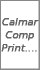
VISUALIZATION _VISU_CTsFlow  // 40x70
VAR_IN_OUT
	m_Inst  : FB_PrintOverview;
END_VAR
    Frame (0,0 40x70), invisible if: m_Inst.aCTV[30]._hidden
        shows CalmarCompPrint._VISU_ContainerView(m_Inst := m_Inst.aCTV[30])
        p3560616238: m_Inst.aCTV[30]._posX
        p2738717112: m_Inst.aCTV[30]._posY
    Frame (0,0 40x70), invisible if: m_Inst.aCTV[31]._hidden
        shows CalmarCompPrint._VISU_ContainerView(m_Inst := m_Inst.aCTV[31])
        p3560616238: m_Inst.aCTV[31]._posX
        p2738717112: m_Inst.aCTV[31]._posY
    Frame (0,0 40x70), invisible if: m_Inst.aCTV[32]._hidden
        shows CalmarCompPrint._VISU_ContainerView(m_Inst := m_Inst.aCTV[32])
        p3560616238: m_Inst.aCTV[32]._posX
        p2738717112: m_Inst.aCTV[32]._posY
    Frame (0,0 40x70), invisible if: m_Inst.aCTV[33]._hidden
        shows CalmarCompPrint._VISU_ContainerView(m_Inst := m_Inst.aCTV[33])
        p3560616238: m_Inst.aCTV[33]._posX
        p2738717112: m_Inst.aCTV[33]._posY
    Frame (0,0 40x70), invisible if: m_Inst.aCTV[34]._hidden
        shows CalmarCompPrint._VISU_ContainerView(m_Inst := m_Inst.aCTV[34])
        p3560616238: m_Inst.aCTV[34]._posX
        p2738717112: m_Inst.aCTV[34]._posY
    Frame (0,0 40x70), invisible if: m_Inst.aCTV[35]._hidden
        shows CalmarCompPrint._VISU_ContainerView(m_Inst := m_Inst.aCTV[35])
        p3560616238: m_Inst.aCTV[35]._posX
        p2738717112: m_Inst.aCTV[35]._posY
    Frame (0,0 40x70), invisible if: m_Inst.aCTV[36]._hidden
        shows CalmarCompPrint._VISU_ContainerView(m_Inst := m_Inst.aCTV[36])
        p3560616238: m_Inst.aCTV[36]._posX
        p2738717112: m_Inst.aCTV[36]._posY
    Frame (0,0 40x70), invisible if: m_Inst.aCTV[37]._hidden
        shows CalmarCompPrint._VISU_ContainerView(m_Inst := m_Inst.aCTV[37])
        p3560616238: m_Inst.aCTV[37]._posX
        p2738717112: m_Inst.aCTV[37]._posY
    Frame (0,0 40x70), invisible if: m_Inst.aCTV[38]._hidden
        shows CalmarCompPrint._VISU_ContainerView(m_Inst := m_Inst.aCTV[38])
        p3560616238: m_Inst.aCTV[38]._posX
        p2738717112: m_Inst.aCTV[38]._posY
    Frame (0,0 40x70), invisible if: m_Inst.aCTV[39]._hidden
        shows CalmarCompPrint._VISU_ContainerView(m_Inst := m_Inst.aCTV[39])
        p3560616238: m_Inst.aCTV[39]._posX
        p2738717112: m_Inst.aCTV[39]._posY
    Frame (0,0 40x70), invisible if: m_Inst.aCTV[10]._hidden
        shows CalmarCompPrint._VISU_ContainerView(m_Inst := m_Inst.aCTV[10])
        p3560616238: m_Inst.aCTV[10]._posX
        p2738717112: m_Inst.aCTV[10]._posY
    Frame (0,0 40x70), invisible if: m_Inst.aCTV[11]._hidden
        shows CalmarCompPrint._VISU_ContainerView(m_Inst := m_Inst.aCTV[11])
        p3560616238: m_Inst.aCTV[11]._posX
        p2738717112: m_Inst.aCTV[11]._posY
    Frame (0,0 40x70), invisible if: m_Inst.aCTV[12]._hidden
        shows CalmarCompPrint._VISU_ContainerView(m_Inst := m_Inst.aCTV[12])
        p3560616238: m_Inst.aCTV[12]._posX
        p2738717112: m_Inst.aCTV[12]._posY
    Frame (0,0 40x70), invisible if: m_Inst.aCTV[13]._hidden
        shows CalmarCompPrint._VISU_ContainerView(m_Inst := m_Inst.aCTV[13])
        p3560616238: m_Inst.aCTV[13]._posX
        p2738717112: m_Inst.aCTV[13]._posY
    Frame (0,0 40x70), invisible if: m_Inst.aCTV[14]._hidden
        shows CalmarCompPrint._VISU_ContainerView(m_Inst := m_Inst.aCTV[14])
        p3560616238: m_Inst.aCTV[14]._posX
        p2738717112: m_Inst.aCTV[14]._posY
    Frame (0,0 40x70), invisible if: m_Inst.aCTV[15]._hidden
        shows CalmarCompPrint._VISU_ContainerView(m_Inst := m_Inst.aCTV[15])
        p3560616238: m_Inst.aCTV[15]._posX
        p2738717112: m_Inst.aCTV[15]._posY
    Frame (0,0 40x70), invisible if: m_Inst.aCTV[16]._hidden
        shows CalmarCompPrint._VISU_ContainerView(m_Inst := m_Inst.aCTV[16])
        p3560616238: m_Inst.aCTV[16]._posX
        p2738717112: m_Inst.aCTV[16]._posY
    Frame (0,0 40x70), invisible if: m_Inst.aCTV[17]._hidden
        shows CalmarCompPrint._VISU_ContainerView(m_Inst := m_Inst.aCTV[17])
        p3560616238: m_Inst.aCTV[17]._posX
        p2738717112: m_Inst.aCTV[17]._posY
    Frame (0,0 40x70), invisible if: m_Inst.aCTV[18]._hidden
        shows CalmarCompPrint._VISU_ContainerView(m_Inst := m_Inst.aCTV[18])
        p3560616238: m_Inst.aCTV[18]._posX
        p2738717112: m_Inst.aCTV[18]._posY
    Frame (0,0 40x70), invisible if: m_Inst.aCTV[19]._hidden
        shows CalmarCompPrint._VISU_ContainerView(m_Inst := m_Inst.aCTV[19])
        p3560616238: m_Inst.aCTV[19]._posX
        p2738717112: m_Inst.aCTV[19]._posY
    Frame (0,0 40x70), invisible if: m_Inst.aCTV[20]._hidden
        shows CalmarCompPrint._VISU_ContainerView(m_Inst := m_Inst.aCTV[20])
        p3560616238: m_Inst.aCTV[20]._posX
        p2738717112: m_Inst.aCTV[20]._posY
    Frame (0,0 40x70), invisible if: m_Inst.aCTV[21]._hidden
        shows CalmarCompPrint._VISU_ContainerView(m_Inst := m_Inst.aCTV[21])
        p3560616238: m_Inst.aCTV[21]._posX
        p2738717112: m_Inst.aCTV[21]._posY
    Frame (0,0 40x70), invisible if: m_Inst.aCTV[22]._hidden
        shows CalmarCompPrint._VISU_ContainerView(m_Inst := m_Inst.aCTV[22])
        p3560616238: m_Inst.aCTV[22]._posX
        p2738717112: m_Inst.aCTV[22]._posY
    Frame (0,0 40x70), invisible if: m_Inst.aCTV[23]._hidden
        shows CalmarCompPrint._VISU_ContainerView(m_Inst := m_Inst.aCTV[23])
        p3560616238: m_Inst.aCTV[23]._posX
        p2738717112: m_Inst.aCTV[23]._posY
    Frame (0,0 40x70), invisible if: m_Inst.aCTV[24]._hidden
        shows CalmarCompPrint._VISU_ContainerView(m_Inst := m_Inst.aCTV[24])
        p3560616238: m_Inst.aCTV[24]._posX
        p2738717112: m_Inst.aCTV[24]._posY
    Frame (0,0 40x70), invisible if: m_Inst.aCTV[25]._hidden
        shows CalmarCompPrint._VISU_ContainerView(m_Inst := m_Inst.aCTV[25])
        p3560616238: m_Inst.aCTV[25]._posX
        p2738717112: m_Inst.aCTV[25]._posY
    Frame (0,0 40x70), invisible if: m_Inst.aCTV[26]._hidden
        shows CalmarCompPrint._VISU_ContainerView(m_Inst := m_Inst.aCTV[26])
        p3560616238: m_Inst.aCTV[26]._posX
        p2738717112: m_Inst.aCTV[26]._posY
    Frame (0,0 40x70), invisible if: m_Inst.aCTV[27]._hidden
        shows CalmarCompPrint._VISU_ContainerView(m_Inst := m_Inst.aCTV[27])
        p3560616238: m_Inst.aCTV[27]._posX
        p2738717112: m_Inst.aCTV[27]._posY
    Frame (0,0 40x70), invisible if: m_Inst.aCTV[28]._hidden
        shows CalmarCompPrint._VISU_ContainerView(m_Inst := m_Inst.aCTV[28])
        p3560616238: m_Inst.aCTV[28]._posX
        p2738717112: m_Inst.aCTV[28]._posY
    Frame (0,0 40x70), invisible if: m_Inst.aCTV[29]._hidden
        shows CalmarCompPrint._VISU_ContainerView(m_Inst := m_Inst.aCTV[29])
        p3560616238: m_Inst.aCTV[29]._posX
        p2738717112: m_Inst.aCTV[29]._posY
    Frame (0,0 40x70), invisible if: m_Inst.aCTV[40]._hidden
        shows CalmarCompPrint._VISU_ContainerView(m_Inst := m_Inst.aCTV[40])
        p3560616238: m_Inst.aCTV[40]._posX
        p2738717112: m_Inst.aCTV[40]._posY
    Frame (0,0 40x70), invisible if: m_Inst.aCTV[41]._hidden
        shows CalmarCompPrint._VISU_ContainerView(m_Inst := m_Inst.aCTV[41])
        p3560616238: m_Inst.aCTV[41]._posX
        p2738717112: m_Inst.aCTV[41]._posY
    Frame (0,0 40x70), invisible if: m_Inst.aCTV[42]._hidden
        shows CalmarCompPrint._VISU_ContainerView(m_Inst := m_Inst.aCTV[42])
        p3560616238: m_Inst.aCTV[42]._posX
        p2738717112: m_Inst.aCTV[42]._posY
    Frame (0,0 40x70), invisible if: m_Inst.aCTV[43]._hidden
        shows CalmarCompPrint._VISU_ContainerView(m_Inst := m_Inst.aCTV[43])
        p3560616238: m_Inst.aCTV[43]._posX
        p2738717112: m_Inst.aCTV[43]._posY
    Frame (0,0 40x70), invisible if: m_Inst.aCTV[44]._hidden
        shows CalmarCompPrint._VISU_ContainerView(m_Inst := m_Inst.aCTV[44])
        p3560616238: m_Inst.aCTV[44]._posX
        p2738717112: m_Inst.aCTV[44]._posY
    Frame (0,0 40x70), invisible if: m_Inst.aCTV[45]._hidden
        shows CalmarCompPrint._VISU_ContainerView(m_Inst := m_Inst.aCTV[45])
        p3560616238: m_Inst.aCTV[45]._posX
        p2738717112: m_Inst.aCTV[45]._posY
    Frame (0,0 40x70), invisible if: m_Inst.aCTV[46]._hidden
        shows CalmarCompPrint._VISU_ContainerView(m_Inst := m_Inst.aCTV[46])
        p3560616238: m_Inst.aCTV[46]._posX
        p2738717112: m_Inst.aCTV[46]._posY
    Frame (0,0 40x70), invisible if: m_Inst.aCTV[47]._hidden
        shows CalmarCompPrint._VISU_ContainerView(m_Inst := m_Inst.aCTV[47])
        p3560616238: m_Inst.aCTV[47]._posX
        p2738717112: m_Inst.aCTV[47]._posY
    Frame (0,0 40x70), invisible if: m_Inst.aCTV[48]._hidden
        shows CalmarCompPrint._VISU_ContainerView(m_Inst := m_Inst.aCTV[48])
        p3560616238: m_Inst.aCTV[48]._posX
        p2738717112: m_Inst.aCTV[48]._posY
    Frame (0,0 40x70), invisible if: m_Inst.aCTV[49]._hidden
        shows CalmarCompPrint._VISU_ContainerView(m_Inst := m_Inst.aCTV[49])
        p3560616238: m_Inst.aCTV[49]._posX
        p2738717112: m_Inst.aCTV[49]._posY
    Frame (0,0 40x70), invisible if: m_Inst.aCTV[49]._hidden
        shows CalmarCompPrint._VISU_ContainerView(m_Inst := m_Inst.aCTV[49])
        p3560616238: m_Inst.aCTV[49]._posX
        p2738717112: m_Inst.aCTV[49]._posY
    Frame (0,0 40x70), invisible if: m_Inst.aCTV[1]._hidden
        shows CalmarCompPrint._VISU_ContainerView(m_Inst := m_Inst.aCTV[1])
        p3560616238: m_Inst.aCTV[1]._posX
        p2738717112: m_Inst.aCTV[1]._posY
    Frame (0,0 40x70), invisible if: m_Inst.aCTV[2]._hidden
        shows CalmarCompPrint._VISU_ContainerView(m_Inst := m_Inst.aCTV[2])
        p3560616238: m_Inst.aCTV[2]._posX
        p2738717112: m_Inst.aCTV[2]._posY
    Frame (0,0 40x70), invisible if: m_Inst.aCTV[3]._hidden
        shows CalmarCompPrint._VISU_ContainerView(m_Inst := m_Inst.aCTV[3])
        p3560616238: m_Inst.aCTV[3]._posX
        p2738717112: m_Inst.aCTV[3]._posY
    Frame (0,0 40x70), invisible if: m_Inst.aCTV[4]._hidden
        shows CalmarCompPrint._VISU_ContainerView(m_Inst := m_Inst.aCTV[4])
        p3560616238: m_Inst.aCTV[4]._posX
        p2738717112: m_Inst.aCTV[4]._posY
    Frame (0,0 40x70), invisible if: m_Inst.aCTV[5]._hidden
        shows CalmarCompPrint._VISU_ContainerView(m_Inst := m_Inst.aCTV[5])
        p3560616238: m_Inst.aCTV[5]._posX
        p2738717112: m_Inst.aCTV[5]._posY
    Frame (0,0 40x70), invisible if: m_Inst.aCTV[6]._hidden
        shows CalmarCompPrint._VISU_ContainerView(m_Inst := m_Inst.aCTV[6])
        p3560616238: m_Inst.aCTV[6]._posX
        p2738717112: m_Inst.aCTV[6]._posY
    Frame (0,0 40x70), invisible if: m_Inst.aCTV[7]._hidden
        shows CalmarCompPrint._VISU_ContainerView(m_Inst := m_Inst.aCTV[7])
        p3560616238: m_Inst.aCTV[7]._posX
        p2738717112: m_Inst.aCTV[7]._posY
    Frame (0,0 40x70), invisible if: m_Inst.aCTV[8]._hidden
        shows CalmarCompPrint._VISU_ContainerView(m_Inst := m_Inst.aCTV[8])
        p3560616238: m_Inst.aCTV[8]._posX
        p2738717112: m_Inst.aCTV[8]._posY
    Frame (0,0 40x70), invisible if: m_Inst.aCTV[9]._hidden
        shows CalmarCompPrint._VISU_ContainerView(m_Inst := m_Inst.aCTV[9])
        p3560616238: m_Inst.aCTV[9]._posX
        p2738717112: m_Inst.aCTV[9]._posY
END_VISUALIZATION

// ---- POUs/Print/DefGrid/_VISU_Templates/_VISU_CTTrackerFlow.TcVIS
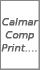
VISUALIZATION _VISU_CTTrackerFlow  // 40x70
VAR_IN_OUT
	m_Inst  : FB_CTTrackerView;
END_VAR
    Frame (0,0 40x70), invisible if: m_Inst.aCTV[30]._hidden
        shows CalmarCompPrint._VISU_ContainerView(m_Inst := m_Inst.aCTV[30])
        p3560616238: m_Inst.aCTV[30]._posX
        p2738717112: m_Inst.aCTV[30]._posY
    Frame (0,0 40x70), invisible if: m_Inst.aCTV[31]._hidden
        shows CalmarCompPrint._VISU_ContainerView(m_Inst := m_Inst.aCTV[31])
        p3560616238: m_Inst.aCTV[31]._posX
        p2738717112: m_Inst.aCTV[31]._posY
    Frame (0,0 40x70), invisible if: m_Inst.aCTV[32]._hidden
        shows CalmarCompPrint._VISU_ContainerView(m_Inst := m_Inst.aCTV[32])
        p3560616238: m_Inst.aCTV[32]._posX
        p2738717112: m_Inst.aCTV[32]._posY
    Frame (0,0 40x70), invisible if: m_Inst.aCTV[33]._hidden
        shows CalmarCompPrint._VISU_ContainerView(m_Inst := m_Inst.aCTV[33])
        p3560616238: m_Inst.aCTV[33]._posX
        p2738717112: m_Inst.aCTV[33]._posY
    Frame (0,0 40x70), invisible if: m_Inst.aCTV[34]._hidden
        shows CalmarCompPrint._VISU_ContainerView(m_Inst := m_Inst.aCTV[34])
        p3560616238: m_Inst.aCTV[34]._posX
        p2738717112: m_Inst.aCTV[34]._posY
    Frame (0,0 40x70), invisible if: m_Inst.aCTV[35]._hidden
        shows CalmarCompPrint._VISU_ContainerView(m_Inst := m_Inst.aCTV[35])
        p3560616238: m_Inst.aCTV[35]._posX
        p2738717112: m_Inst.aCTV[35]._posY
    Frame (0,0 40x70), invisible if: m_Inst.aCTV[36]._hidden
        shows CalmarCompPrint._VISU_ContainerView(m_Inst := m_Inst.aCTV[36])
        p3560616238: m_Inst.aCTV[36]._posX
        p2738717112: m_Inst.aCTV[36]._posY
    Frame (0,0 40x70), invisible if: m_Inst.aCTV[37]._hidden
        shows CalmarCompPrint._VISU_ContainerView(m_Inst := m_Inst.aCTV[37])
        p3560616238: m_Inst.aCTV[37]._posX
        p2738717112: m_Inst.aCTV[37]._posY
    Frame (0,0 40x70), invisible if: m_Inst.aCTV[38]._hidden
        shows CalmarCompPrint._VISU_ContainerView(m_Inst := m_Inst.aCTV[38])
        p3560616238: m_Inst.aCTV[38]._posX
        p2738717112: m_Inst.aCTV[38]._posY
    Frame (0,0 40x70), invisible if: m_Inst.aCTV[39]._hidden
        shows CalmarCompPrint._VISU_ContainerView(m_Inst := m_Inst.aCTV[39])
        p3560616238: m_Inst.aCTV[39]._posX
        p2738717112: m_Inst.aCTV[39]._posY
    Frame (0,0 40x70), invisible if: m_Inst.aCTV[10]._hidden
        shows CalmarCompPrint._VISU_ContainerView(m_Inst := m_Inst.aCTV[10])
        p3560616238: m_Inst.aCTV[10]._posX
        p2738717112: m_Inst.aCTV[10]._posY
    Frame (0,0 40x70), invisible if: m_Inst.aCTV[11]._hidden
        shows CalmarCompPrint._VISU_ContainerView(m_Inst := m_Inst.aCTV[11])
        p3560616238: m_Inst.aCTV[11]._posX
        p2738717112: m_Inst.aCTV[11]._posY
    Frame (0,0 40x70), invisible if: m_Inst.aCTV[12]._hidden
        shows CalmarCompPrint._VISU_ContainerView(m_Inst := m_Inst.aCTV[12])
        p3560616238: m_Inst.aCTV[12]._posX
        p2738717112: m_Inst.aCTV[12]._posY
    Frame (0,0 40x70), invisible if: m_Inst.aCTV[13]._hidden
        shows CalmarCompPrint._VISU_ContainerView(m_Inst := m_Inst.aCTV[13])
        p3560616238: m_Inst.aCTV[13]._posX
        p2738717112: m_Inst.aCTV[13]._posY
    Frame (0,0 40x70), invisible if: m_Inst.aCTV[14]._hidden
        shows CalmarCompPrint._VISU_ContainerView(m_Inst := m_Inst.aCTV[14])
        p3560616238: m_Inst.aCTV[14]._posX
        p2738717112: m_Inst.aCTV[14]._posY
    Frame (0,0 40x70), invisible if: m_Inst.aCTV[15]._hidden
        shows CalmarCompPrint._VISU_ContainerView(m_Inst := m_Inst.aCTV[15])
        p3560616238: m_Inst.aCTV[15]._posX
        p2738717112: m_Inst.aCTV[15]._posY
    Frame (0,0 40x70), invisible if: m_Inst.aCTV[16]._hidden
        shows CalmarCompPrint._VISU_ContainerView(m_Inst := m_Inst.aCTV[16])
        p3560616238: m_Inst.aCTV[16]._posX
        p2738717112: m_Inst.aCTV[16]._posY
    Frame (0,0 40x70), invisible if: m_Inst.aCTV[17]._hidden
        shows CalmarCompPrint._VISU_ContainerView(m_Inst := m_Inst.aCTV[17])
        p3560616238: m_Inst.aCTV[17]._posX
        p2738717112: m_Inst.aCTV[17]._posY
    Frame (0,0 40x70), invisible if: m_Inst.aCTV[18]._hidden
        shows CalmarCompPrint._VISU_ContainerView(m_Inst := m_Inst.aCTV[18])
        p3560616238: m_Inst.aCTV[18]._posX
        p2738717112: m_Inst.aCTV[18]._posY
    Frame (0,0 40x70), invisible if: m_Inst.aCTV[19]._hidden
        shows CalmarCompPrint._VISU_ContainerView(m_Inst := m_Inst.aCTV[19])
        p3560616238: m_Inst.aCTV[19]._posX
        p2738717112: m_Inst.aCTV[19]._posY
    Frame (0,0 40x70), invisible if: m_Inst.aCTV[20]._hidden
        shows CalmarCompPrint._VISU_ContainerView(m_Inst := m_Inst.aCTV[20])
        p3560616238: m_Inst.aCTV[20]._posX
        p2738717112: m_Inst.aCTV[20]._posY
    Frame (0,0 40x70), invisible if: m_Inst.aCTV[21]._hidden
        shows CalmarCompPrint._VISU_ContainerView(m_Inst := m_Inst.aCTV[21])
        p3560616238: m_Inst.aCTV[21]._posX
        p2738717112: m_Inst.aCTV[21]._posY
    Frame (0,0 40x70), invisible if: m_Inst.aCTV[22]._hidden
        shows CalmarCompPrint._VISU_ContainerView(m_Inst := m_Inst.aCTV[22])
        p3560616238: m_Inst.aCTV[22]._posX
        p2738717112: m_Inst.aCTV[22]._posY
    Frame (0,0 40x70), invisible if: m_Inst.aCTV[23]._hidden
        shows CalmarCompPrint._VISU_ContainerView(m_Inst := m_Inst.aCTV[23])
        p3560616238: m_Inst.aCTV[23]._posX
        p2738717112: m_Inst.aCTV[23]._posY
    Frame (0,0 40x70), invisible if: m_Inst.aCTV[24]._hidden
        shows CalmarCompPrint._VISU_ContainerView(m_Inst := m_Inst.aCTV[24])
        p3560616238: m_Inst.aCTV[24]._posX
        p2738717112: m_Inst.aCTV[24]._posY
    Frame (0,0 40x70), invisible if: m_Inst.aCTV[25]._hidden
        shows CalmarCompPrint._VISU_ContainerView(m_Inst := m_Inst.aCTV[25])
        p3560616238: m_Inst.aCTV[25]._posX
        p2738717112: m_Inst.aCTV[25]._posY
    Frame (0,0 40x70), invisible if: m_Inst.aCTV[26]._hidden
        shows CalmarCompPrint._VISU_ContainerView(m_Inst := m_Inst.aCTV[26])
        p3560616238: m_Inst.aCTV[26]._posX
        p2738717112: m_Inst.aCTV[26]._posY
    Frame (0,0 40x70), invisible if: m_Inst.aCTV[27]._hidden
        shows CalmarCompPrint._VISU_ContainerView(m_Inst := m_Inst.aCTV[27])
        p3560616238: m_Inst.aCTV[27]._posX
        p2738717112: m_Inst.aCTV[27]._posY
    Frame (0,0 40x70), invisible if: m_Inst.aCTV[28]._hidden
        shows CalmarCompPrint._VISU_ContainerView(m_Inst := m_Inst.aCTV[28])
        p3560616238: m_Inst.aCTV[28]._posX
        p2738717112: m_Inst.aCTV[28]._posY
    Frame (0,0 40x70), invisible if: m_Inst.aCTV[29]._hidden
        shows CalmarCompPrint._VISU_ContainerView(m_Inst := m_Inst.aCTV[29])
        p3560616238: m_Inst.aCTV[29]._posX
        p2738717112: m_Inst.aCTV[29]._posY
    Frame (0,0 40x70), invisible if: m_Inst.aCTV[40]._hidden
        shows CalmarCompPrint._VISU_ContainerView(m_Inst := m_Inst.aCTV[40])
        p3560616238: m_Inst.aCTV[40]._posX
        p2738717112: m_Inst.aCTV[40]._posY
    Frame (0,0 40x70), invisible if: m_Inst.aCTV[41]._hidden
        shows CalmarCompPrint._VISU_ContainerView(m_Inst := m_Inst.aCTV[41])
        p3560616238: m_Inst.aCTV[41]._posX
        p2738717112: m_Inst.aCTV[41]._posY
    Frame (0,0 40x70), invisible if: m_Inst.aCTV[42]._hidden
        shows CalmarCompPrint._VISU_ContainerView(m_Inst := m_Inst.aCTV[42])
        p3560616238: m_Inst.aCTV[42]._posX
        p2738717112: m_Inst.aCTV[42]._posY
    Frame (0,0 40x70), invisible if: m_Inst.aCTV[43]._hidden
        shows CalmarCompPrint._VISU_ContainerView(m_Inst := m_Inst.aCTV[43])
        p3560616238: m_Inst.aCTV[43]._posX
        p2738717112: m_Inst.aCTV[43]._posY
    Frame (0,0 40x70), invisible if: m_Inst.aCTV[44]._hidden
        shows CalmarCompPrint._VISU_ContainerView(m_Inst := m_Inst.aCTV[44])
        p3560616238: m_Inst.aCTV[44]._posX
        p2738717112: m_Inst.aCTV[44]._posY
    Frame (0,0 40x70), invisible if: m_Inst.aCTV[45]._hidden
        shows CalmarCompPrint._VISU_ContainerView(m_Inst := m_Inst.aCTV[45])
        p3560616238: m_Inst.aCTV[45]._posX
        p2738717112: m_Inst.aCTV[45]._posY
    Frame (0,0 40x70), invisible if: m_Inst.aCTV[46]._hidden
        shows CalmarCompPrint._VISU_ContainerView(m_Inst := m_Inst.aCTV[46])
        p3560616238: m_Inst.aCTV[46]._posX
        p2738717112: m_Inst.aCTV[46]._posY
    Frame (0,0 40x70), invisible if: m_Inst.aCTV[47]._hidden
        shows CalmarCompPrint._VISU_ContainerView(m_Inst := m_Inst.aCTV[47])
        p3560616238: m_Inst.aCTV[47]._posX
        p2738717112: m_Inst.aCTV[47]._posY
    Frame (0,0 40x70), invisible if: m_Inst.aCTV[48]._hidden
        shows CalmarCompPrint._VISU_ContainerView(m_Inst := m_Inst.aCTV[48])
        p3560616238: m_Inst.aCTV[48]._posX
        p2738717112: m_Inst.aCTV[48]._posY
    Frame (0,0 40x70), invisible if: m_Inst.aCTV[49]._hidden
        shows CalmarCompPrint._VISU_ContainerView(m_Inst := m_Inst.aCTV[49])
        p3560616238: m_Inst.aCTV[49]._posX
        p2738717112: m_Inst.aCTV[49]._posY
    Frame (0,0 40x70), invisible if: m_Inst.aCTV[49]._hidden
        shows CalmarCompPrint._VISU_ContainerView(m_Inst := m_Inst.aCTV[49])
        p3560616238: m_Inst.aCTV[49]._posX
        p2738717112: m_Inst.aCTV[49]._posY
    Frame (0,0 40x70), invisible if: m_Inst.aCTV[1]._hidden
        shows CalmarCompPrint._VISU_ContainerView(m_Inst := m_Inst.aCTV[1])
        p3560616238: m_Inst.aCTV[1]._posX
        p2738717112: m_Inst.aCTV[1]._posY
    Frame (0,0 40x70), invisible if: m_Inst.aCTV[2]._hidden
        shows CalmarCompPrint._VISU_ContainerView(m_Inst := m_Inst.aCTV[2])
        p3560616238: m_Inst.aCTV[2]._posX
        p2738717112: m_Inst.aCTV[2]._posY
    Frame (0,0 40x70), invisible if: m_Inst.aCTV[3]._hidden
        shows CalmarCompPrint._VISU_ContainerView(m_Inst := m_Inst.aCTV[3])
        p3560616238: m_Inst.aCTV[3]._posX
        p2738717112: m_Inst.aCTV[3]._posY
    Frame (0,0 40x70), invisible if: m_Inst.aCTV[4]._hidden
        shows CalmarCompPrint._VISU_ContainerView(m_Inst := m_Inst.aCTV[4])
        p3560616238: m_Inst.aCTV[4]._posX
        p2738717112: m_Inst.aCTV[4]._posY
    Frame (0,0 40x70), invisible if: m_Inst.aCTV[5]._hidden
        shows CalmarCompPrint._VISU_ContainerView(m_Inst := m_Inst.aCTV[5])
        p3560616238: m_Inst.aCTV[5]._posX
        p2738717112: m_Inst.aCTV[5]._posY
    Frame (0,0 40x70), invisible if: m_Inst.aCTV[6]._hidden
        shows CalmarCompPrint._VISU_ContainerView(m_Inst := m_Inst.aCTV[6])
        p3560616238: m_Inst.aCTV[6]._posX
        p2738717112: m_Inst.aCTV[6]._posY
    Frame (0,0 40x70), invisible if: m_Inst.aCTV[7]._hidden
        shows CalmarCompPrint._VISU_ContainerView(m_Inst := m_Inst.aCTV[7])
        p3560616238: m_Inst.aCTV[7]._posX
        p2738717112: m_Inst.aCTV[7]._posY
    Frame (0,0 40x70), invisible if: m_Inst.aCTV[8]._hidden
        shows CalmarCompPrint._VISU_ContainerView(m_Inst := m_Inst.aCTV[8])
        p3560616238: m_Inst.aCTV[8]._posX
        p2738717112: m_Inst.aCTV[8]._posY
    Frame (0,0 40x70), invisible if: m_Inst.aCTV[9]._hidden
        shows CalmarCompPrint._VISU_ContainerView(m_Inst := m_Inst.aCTV[9])
        p3560616238: m_Inst.aCTV[9]._posX
        p2738717112: m_Inst.aCTV[9]._posY
END_VISUALIZATION

// ---- POUs/Print/DefGrid/_VISU_Templates/_VISU_CT_Details.TcVIS
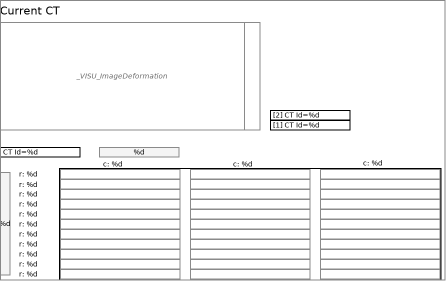
VISUALIZATION _VISU_CT_Details  // 446x281
VAR_IN_OUT
  mInst : FB_WorkerDefGrid;
END_VAR
    Frame (0,22 260x108)
        shows _VISU_ContainerDefGrid(m_Inst := mInst._pAttachedCt^)
    Frame (16,159 427x122)
        shows _VISU_DefGridTable(m_Inst := mInst._pAttachedCt^.fBImageDeformation, m_row_start := mInst.nGridRowStart, m_col_start := mInst.nGridColStart)
    Scrollbar (99,147 80x10), "%d", text variable: mInst.nGridColStart
        p2245068023: mInst._pAttachedCt^.fBImageDeformation.nMAX_ROWS_DEFGRID-2
        p1057716461: mInst.nGridColStart
    Scrollbar (0,172 10x103), "%d", text variable: mInst._pAttachedCt^.sContainer.iId
        p2245068023: mInst._pAttachedCt^.fBImageDeformation.nMAX_ROWS_DEFGRID
        p1057716461: mInst.nGridRowStart
    Label (-3,1 150x20), "Current CT"
    Rectangle (0,147 80x10), "CT Id=%d", text variable: mInst._pAttachedCt^.sContainer.iId
    Rectangle (270,120 80x10), "[1] CT Id=%d", text variable: mInst._pAttachedCTList[1]^.sContainer.iId, input disabled if: mInst._pAttachedCTList[1] = 0
    Rectangle (270,110 80x10), "[2] CT Id=%d", text variable: mInst._pAttachedCTList[1]^.sContainer.iId, invisible if: mInst._pAttachedCTList[2] = 0, input disabled if: mInst._pAttachedCTList[1] = 0
END_VISUALIZATION

// ---- POUs/Print/DefGrid/_VISU_Templates/_VISU_DefGridTable.TcVIS
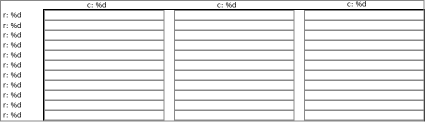
VISUALIZATION _VISU_DefGridTable  // 425x122
VAR_IN_OUT
	m_Inst : FB_ImageDeformation;
  m_row_start : UDINT;
  m_col_start : UDINT;
END_VAR
    Rectangle (43,9 382x112)
    Frame (44,10 120x10)
        shows _VISU_GridPointView(m_Inst := m_Inst._sDefGridPoints[0+m_col_start, 0+m_row_start])
    Frame (44,20 120x10)
        shows _VISU_GridPointView(m_Inst := m_Inst._sDefGridPoints[0+m_col_start, 1+m_row_start])
    Frame (44,30 120x10)
        shows _VISU_GridPointView(m_Inst := m_Inst._sDefGridPoints[0+m_col_start, 2+m_row_start])
    Frame (44,40 120x10)
        shows _VISU_GridPointView(m_Inst := m_Inst._sDefGridPoints[0+m_col_start, 3+m_row_start])
    Frame (44,50 120x10)
        shows _VISU_GridPointView(m_Inst := m_Inst._sDefGridPoints[0+m_col_start, 4+m_row_start])
    Frame (44,60 120x10)
        shows _VISU_GridPointView(m_Inst := m_Inst._sDefGridPoints[0+m_col_start, 5+m_row_start])
    Frame (44,70 120x10)
        shows _VISU_GridPointView(m_Inst := m_Inst._sDefGridPoints[0+m_col_start, 6+m_row_start])
    Frame (44,80 120x10)
        shows _VISU_GridPointView(m_Inst := m_Inst._sDefGridPoints[0+m_col_start, 7+m_row_start])
    Frame (44,90 120x10)
        shows _VISU_GridPointView(m_Inst := m_Inst._sDefGridPoints[0+m_col_start, 8+m_row_start])
    Frame (44,100 120x10)
        shows _VISU_GridPointView(m_Inst := m_Inst._sDefGridPoints[0+m_col_start, 9+m_row_start])
    Frame (44,110 120x10)
        shows _VISU_GridPointView(m_Inst := m_Inst._sDefGridPoints[0+m_col_start, 10+m_row_start])
    Frame (174,10 120x10)
        shows _VISU_GridPointView(m_Inst := m_Inst._sDefGridPoints[1+m_col_start, 0+m_row_start])
    Frame (174,20 120x10)
        shows _VISU_GridPointView(m_Inst := m_Inst._sDefGridPoints[1+m_col_start, 1+m_row_start])
    Frame (174,30 120x10)
        shows _VISU_GridPointView(m_Inst := m_Inst._sDefGridPoints[1+m_col_start, 2+m_row_start])
    Frame (174,40 120x10)
        shows _VISU_GridPointView(m_Inst := m_Inst._sDefGridPoints[1+m_col_start, 3+m_row_start])
    Frame (174,50 120x10)
        shows _VISU_GridPointView(m_Inst := m_Inst._sDefGridPoints[1+m_col_start, 4+m_row_start])
    Frame (174,60 120x10)
        shows _VISU_GridPointView(m_Inst := m_Inst._sDefGridPoints[1+m_col_start, 5+m_row_start])
    Frame (174,70 120x10)
        shows _VISU_GridPointView(m_Inst := m_Inst._sDefGridPoints[1+m_col_start, 6+m_row_start])
    Frame (174,80 120x10)
        shows _VISU_GridPointView(m_Inst := m_Inst._sDefGridPoints[1+m_col_start, 7+m_row_start])
    Frame (174,90 120x10)
        shows _VISU_GridPointView(m_Inst := m_Inst._sDefGridPoints[1+m_col_start, 8+m_row_start])
    Frame (174,100 120x10)
        shows _VISU_GridPointView(m_Inst := m_Inst._sDefGridPoints[1+m_col_start, 9+m_row_start])
    Frame (174,110 120x10)
        shows _VISU_GridPointView(m_Inst := m_Inst._sDefGridPoints[1+m_col_start, 10+m_row_start])
    Frame (304,10 120x10)
        shows _VISU_GridPointView(m_Inst := m_Inst._sDefGridPoints[2+m_col_start, 0+m_row_start])
    Frame (304,20 120x10)
        shows _VISU_GridPointView(m_Inst := m_Inst._sDefGridPoints[2+m_col_start, 1+m_row_start])
    Frame (304,30 120x10)
        shows _VISU_GridPointView(m_Inst := m_Inst._sDefGridPoints[2+m_col_start, 2+m_row_start])
    Frame (304,40 120x10)
        shows _VISU_GridPointView(m_Inst := m_Inst._sDefGridPoints[2+m_col_start, 3+m_row_start])
    Frame (304,50 120x10)
        shows _VISU_GridPointView(m_Inst := m_Inst._sDefGridPoints[2+m_col_start, 4+m_row_start])
    Frame (304,60 120x10)
        shows _VISU_GridPointView(m_Inst := m_Inst._sDefGridPoints[2+m_col_start, 5+m_row_start])
    Frame (304,70 120x10)
        shows _VISU_GridPointView(m_Inst := m_Inst._sDefGridPoints[2+m_col_start, 6+m_row_start])
    Frame (304,80 120x10)
        shows _VISU_GridPointView(m_Inst := m_Inst._sDefGridPoints[2+m_col_start, 7+m_row_start])
    Frame (304,90 120x10)
        shows _VISU_GridPointView(m_Inst := m_Inst._sDefGridPoints[2+m_col_start, 8+m_row_start])
    Frame (304,100 120x10)
        shows _VISU_GridPointView(m_Inst := m_Inst._sDefGridPoints[2+m_col_start, 9+m_row_start])
    Frame (304,110 120x10)
        shows _VISU_GridPointView(m_Inst := m_Inst._sDefGridPoints[2+m_col_start, 10+m_row_start])
    Rectangle (84,0 40x10), "c: %d", text variable: m_col_start
    Rectangle (214,0 40x10), "c: %d", text variable: m_col_start+1
    Rectangle (344,-1 40x10), "c: %d", text variable: m_col_start+2
    Rectangle (0,10 40x10), "r: %d", text variable: m_row_start
    Rectangle (0,20 40x11), "r: %d", text variable: m_row_start+1
    Rectangle (0,30 40x10), "r: %d", text variable: m_row_start+2
    Rectangle (0,40 40x10), "r: %d", text variable: m_row_start+3
    Rectangle (0,50 40x10), "r: %d", text variable: m_row_start+4
    Rectangle (0,60 40x10), "r: %d", text variable: m_row_start+5
    Rectangle (0,70 40x10), "r: %d", text variable: m_row_start+6
    Rectangle (0,80 40x10), "r: %d", text variable: m_row_start+7
    Rectangle (0,90 40x10), "r: %d", text variable: m_row_start+8
    Rectangle (0,100 40x10), "r: %d", text variable: m_row_start+9
    Rectangle (0,110 40x10), "r: %d", text variable: m_row_start+10
END_VISUALIZATION

// ---- POUs/Print/DefGrid/_VISU_Templates/_VISU_DefGridTable_raw.TcVIS
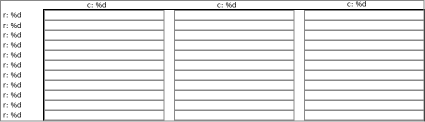
VISUALIZATION _VISU_DefGridTable_raw  // 425x122
VAR_IN_OUT
	mGridTable : ARRAY[0..100, 0..100] OF ST_DeformationPointTbl;
  mGridRowStart : UDINT;
  mGridColStart : UDINT;
END_VAR
    Rectangle (43,9 382x112)
    Frame (44,10 120x10)
        shows _VISU_GridPointView(mGridTable := mGridTable[0+mGridColStart, 0+mGridRowStart])
        pReferences[0]: mGridTable=mGridTable[0+mGridColStart, 0+mGridRowStart]
    Frame (44,20 120x10)
        shows _VISU_GridPointView(mGridTable := mGridTable[0+mGridColStart, 1+mGridRowStart])
        pReferences[0]: mGridTable=mGridTable[0+mGridColStart, 1+mGridRowStart]
    Frame (44,30 120x10)
        shows _VISU_GridPointView(mGridTable := mGridTable[0+mGridColStart, 2+mGridRowStart])
        pReferences[0]: mGridTable=mGridTable[0+mGridColStart, 2+mGridRowStart]
    Frame (44,40 120x10)
        shows _VISU_GridPointView(mGridTable := mGridTable[0+mGridColStart, 3+mGridRowStart])
        pReferences[0]: mGridTable=mGridTable[0+mGridColStart, 3+mGridRowStart]
    Frame (44,50 120x10)
        shows _VISU_GridPointView(mGridTable := mGridTable[0+mGridColStart, 4+mGridRowStart])
        pReferences[0]: mGridTable=mGridTable[0+mGridColStart, 4+mGridRowStart]
    Frame (44,60 120x10)
        shows _VISU_GridPointView(mGridTable := mGridTable[0+mGridColStart, 5+mGridRowStart])
        pReferences[0]: mGridTable=mGridTable[0+mGridColStart, 5+mGridRowStart]
    Frame (44,70 120x10)
        shows _VISU_GridPointView(mGridTable := mGridTable[0+mGridColStart, 6+mGridRowStart])
        pReferences[0]: mGridTable=mGridTable[0+mGridColStart, 6+mGridRowStart]
    Frame (44,80 120x10)
        shows _VISU_GridPointView(mGridTable := mGridTable[0+mGridColStart, 7+mGridRowStart])
        pReferences[0]: mGridTable=mGridTable[0+mGridColStart, 7+mGridRowStart]
    Frame (44,90 120x10)
        shows _VISU_GridPointView(mGridTable := mGridTable[0+mGridColStart, 8+mGridRowStart])
        pReferences[0]: mGridTable=mGridTable[0+mGridColStart, 8+mGridRowStart]
    Frame (44,100 120x10)
        shows _VISU_GridPointView(mGridTable := mGridTable[0+mGridColStart, 9+mGridRowStart])
        pReferences[0]: mGridTable=mGridTable[0+mGridColStart, 9+mGridRowStart]
    Frame (44,110 120x10)
        shows _VISU_GridPointView(mGridTable := mGridTable[0+mGridColStart, 10+mGridRowStart])
        pReferences[0]: mGridTable=mGridTable[0+mGridColStart, 10+mGridRowStart]
    Frame (174,10 120x10)
        shows _VISU_GridPointView(mGridTable := mGridTable[1+mGridColStart, 0+mGridRowStart])
        pReferences[0]: mGridTable=mGridTable[1+mGridColStart, 0+mGridRowStart]
    Frame (174,20 120x10)
        shows _VISU_GridPointView(mGridTable := mGridTable[1+mGridColStart, 1+mGridRowStart])
        pReferences[0]: mGridTable=mGridTable[1+mGridColStart, 1+mGridRowStart]
    Frame (174,30 120x10)
        shows _VISU_GridPointView(mGridTable := mGridTable[1+mGridColStart, 2+mGridRowStart])
        pReferences[0]: mGridTable=mGridTable[1+mGridColStart, 2+mGridRowStart]
    Frame (174,40 120x10)
        shows _VISU_GridPointView(mGridTable := mGridTable[1+mGridColStart, 3+mGridRowStart])
        pReferences[0]: mGridTable=mGridTable[1+mGridColStart, 3+mGridRowStart]
    Frame (174,50 120x10)
        shows _VISU_GridPointView(mGridTable := mGridTable[1+mGridColStart, 4+mGridRowStart])
        pReferences[0]: mGridTable=mGridTable[1+mGridColStart, 4+mGridRowStart]
    Frame (174,60 120x10)
        shows _VISU_GridPointView(mGridTable := mGridTable[1+mGridColStart, 5+mGridRowStart])
        pReferences[0]: mGridTable=mGridTable[1+mGridColStart, 5+mGridRowStart]
    Frame (174,70 120x10)
        shows _VISU_GridPointView(mGridTable := mGridTable[1+mGridColStart, 6+mGridRowStart])
        pReferences[0]: mGridTable=mGridTable[1+mGridColStart, 6+mGridRowStart]
    Frame (174,80 120x10)
        shows _VISU_GridPointView(mGridTable := mGridTable[1+mGridColStart, 7+mGridRowStart])
        pReferences[0]: mGridTable=mGridTable[1+mGridColStart, 7+mGridRowStart]
    Frame (174,90 120x10)
        shows _VISU_GridPointView(mGridTable := mGridTable[1+mGridColStart, 8+mGridRowStart])
        pReferences[0]: mGridTable=mGridTable[1+mGridColStart, 8+mGridRowStart]
    Frame (174,100 120x10)
        shows _VISU_GridPointView(mGridTable := mGridTable[1+mGridColStart, 9+mGridRowStart])
        pReferences[0]: mGridTable=mGridTable[1+mGridColStart, 9+mGridRowStart]
    Frame (174,110 120x10)
        shows _VISU_GridPointView(mGridTable := mGridTable[1+mGridColStart, 10+mGridRowStart])
        pReferences[0]: mGridTable=mGridTable[1+mGridColStart, 10+mGridRowStart]
    Frame (304,10 120x10)
        shows _VISU_GridPointView(mGridTable := mGridTable[2+mGridColStart, 0+mGridRowStart])
        pReferences[0]: mGridTable=mGridTable[2+mGridColStart, 0+mGridRowStart]
    Frame (304,20 120x10)
        shows _VISU_GridPointView(mGridTable := mGridTable[2+mGridColStart, 1+mGridRowStart])
        pReferences[0]: mGridTable=mGridTable[2+mGridColStart, 1+mGridRowStart]
    Frame (304,30 120x10)
        shows _VISU_GridPointView(mGridTable := mGridTable[2+mGridColStart, 2+mGridRowStart])
        pReferences[0]: mGridTable=mGridTable[2+mGridColStart, 2+mGridRowStart]
    Frame (304,40 120x10)
        shows _VISU_GridPointView(mGridTable := mGridTable[2+mGridColStart, 3+mGridRowStart])
        pReferences[0]: mGridTable=mGridTable[2+mGridColStart, 3+mGridRowStart]
    Frame (304,50 120x10)
        shows _VISU_GridPointView(mGridTable := mGridTable[2+mGridColStart, 4+mGridRowStart])
        pReferences[0]: mGridTable=mGridTable[2+mGridColStart, 4+mGridRowStart]
    Frame (304,60 120x10)
        shows _VISU_GridPointView(mGridTable := mGridTable[2+mGridColStart, 5+mGridRowStart])
        pReferences[0]: mGridTable=mGridTable[2+mGridColStart, 5+mGridRowStart]
    Frame (304,70 120x10)
        shows _VISU_GridPointView(mGridTable := mGridTable[2+mGridColStart, 6+mGridRowStart])
        pReferences[0]: mGridTable=mGridTable[2+mGridColStart, 6+mGridRowStart]
    Frame (304,80 120x10)
        shows _VISU_GridPointView(mGridTable := mGridTable[2+mGridColStart, 7+mGridRowStart])
        pReferences[0]: mGridTable=mGridTable[2+mGridColStart, 7+mGridRowStart]
    Frame (304,90 120x10)
        shows _VISU_GridPointView(mGridTable := mGridTable[2+mGridColStart, 8+mGridRowStart])
        pReferences[0]: mGridTable=mGridTable[2+mGridColStart, 8+mGridRowStart]
    Frame (304,100 120x10)
        shows _VISU_GridPointView(mGridTable := mGridTable[2+mGridColStart, 9+mGridRowStart])
        pReferences[0]: mGridTable=mGridTable[2+mGridColStart, 9+mGridRowStart]
    Frame (304,110 120x10)
        shows _VISU_GridPointView(mGridTable := mGridTable[2+mGridColStart, 10+mGridRowStart])
        pReferences[0]: mGridTable=mGridTable[2+mGridColStart, 10+mGridRowStart]
    Rectangle (84,0 40x10), "c: %d", text variable: mGridColStart
    Rectangle (214,0 40x10), "c: %d", text variable: mGridColStart+1
    Rectangle (344,-1 40x10), "c: %d", text variable: mGridColStart+2
    Rectangle (0,10 40x10), "r: %d", text variable: mGridRowStart
    Rectangle (0,20 40x11), "r: %d", text variable: mGridRowStart+1
    Rectangle (0,30 40x10), "r: %d", text variable: mGridRowStart+2
    Rectangle (0,40 40x10), "r: %d", text variable: mGridRowStart+3
    Rectangle (0,50 40x10), "r: %d", text variable: mGridRowStart+4
    Rectangle (0,60 40x10), "r: %d", text variable: mGridRowStart+5
    Rectangle (0,70 40x10), "r: %d", text variable: mGridRowStart+6
    Rectangle (0,80 40x10), "r: %d", text variable: mGridRowStart+7
    Rectangle (0,90 40x10), "r: %d", text variable: mGridRowStart+8
    Rectangle (0,100 40x10), "r: %d", text variable: mGridRowStart+9
    Rectangle (0,110 40x10), "r: %d", text variable: mGridRowStart+10
END_VISUALIZATION

// ---- POUs/Print/DefGrid/_VISU_Templates/_VISU_FineAlignment.TcVIS
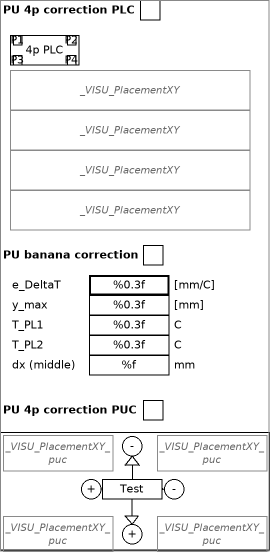
VISUALIZATION _VISU_FineAlignment  // 270x552
VAR_IN_OUT
	mInst : FB_FineAlignement;
END_VAR
    Rectangle (0,432 270x118)
    Rectangle (0,0 259x427)
    Rectangle (0,0 140x20), "PU 4p correction PLC"
    RoundedRectangle (140,0 20x20)
        toggle mInst._bEnable_4p
    Rectangle (0,245 140x20), "PU banana correction"
    RoundedRectangle (143,245 20x20)
        toggle mInst._bEnable_banana
    Rectangle (0,400 140x20), "PU 4p correction PUC"
    RoundedRectangle (143,400 20x20)
        toggle mInst._bEnablePuc_4p
    Frame (10,70 240x40)
        shows _VISU_PlacementXY(m_Inst := mInst._fbPlcCorrPoints[1])
    Group (10,35 69x30)
        RoundedRectangle (0,0 69x30), "4p PLC"
        Rectangle (3,0 9x10), "P1"
        Rectangle (57,0 9x10), "P2"
        Rectangle (57,20 9x10), "P4"
        Rectangle (3,20 9x10), "P3"
    Frame (10,110 240x40)
        shows _VISU_PlacementXY(m_Inst := mInst._fbPlcCorrPoints[2])
    Frame (10,150 240x40)
        shows _VISU_PlacementXY(m_Inst := mInst._fbPlcCorrPoints[3])
    Frame (10,190 240x40)
        shows _VISU_PlacementXY(m_Inst := mInst._fbPlcCorrPoints[4])
    Rectangle (89,275 80x20), "%0.3f", text variable: mInst._e_max_per_deltaT
        OnMouseClick: write the text variable via Default
    Rectangle (89,295 80x20), "%0.3f", text variable: mInst._y_max
    Rectangle (9,275 80x20), "e_DeltaT"
    Rectangle (9,295 80x20), "y_max"
    Rectangle (171,295 51x20), "[mm]"
    Rectangle (171,275 51x20), "[mm/C]"
    Rectangle (89,315 80x20), "%0.3f", text variable: mInst._fT1
    Rectangle (89,335 80x20), "%0.3f", text variable: mInst._fT2
    Rectangle (9,315 80x20), "T_PL1"
    Rectangle (9,335 80x20), "T_PL2"
    Rectangle (171,315 51x20), "C"
    Rectangle (171,335 51x20), "C"
    Rectangle (89,355 80x20), "%f", text variable: mInst._dx_middle
    Rectangle (9,355 80x20), "dx (middle)"
    Rectangle (171,355 51x20), "mm"
    Frame (3,435 110x36)
        shows _VISU_PlacementXY_puc(mInst := mInst._pAdsCam^.stAds.sI_CorrectionPointIndication[1], aName := mInst.aPucPointNames[1], bSelected := mInst.bSelected[1], bSelect := mInst.bSelect[1])
    Frame (157,435 110x36)
        shows _VISU_PlacementXY_puc(mInst := mInst._pAdsCam^.stAds.sI_CorrectionPointIndication[2], aName := mInst.aPucPointNames[2], bSelected := mInst.bSelected[2], bSelect := mInst.bSelect[2])
    Frame (3,516 110x36)
        shows _VISU_PlacementXY_puc(mInst := mInst._pAdsCam^.stAds.sI_CorrectionPointIndication[3], aName := mInst.aPucPointNames[3], bSelected := mInst.bSelected[3], bSelect := mInst.bSelect[3])
    Frame (157,516 110x36)
        shows _VISU_PlacementXY_puc(mInst := mInst._pAdsCam^.stAds.sI_CorrectionPointIndication[4], aName := mInst.aPucPointNames[4], bSelected := mInst.bSelected[4], bSelect := mInst.bSelect[4])
    Group (81,436 103x108), invisible if: NOT mInst._bUT_4pPuc
        Ellipse (41,0 20x20), "-"
            toggle mInst.bYMinus
        Ellipse (41,88 20x20), "+"
            toggle mInst.bYPlus
        Polyline (51,29) (44,29) (51,20) (58,29) (51,29) (51,46)
        Polyline (51,80) (44,80) (51,88) (57,80) (51,80) (51,63)
        Ellipse (83,43 20x20), "-"
            toggle mInst.bXMinus
        Ellipse (0,43 20x20), "+"
            toggle mInst.bXPlus
        Polyline (28,53) (28,47) (21,53) (28,59) (28,53) (44,53)
        Polyline (74,54) (74,46) (82,53) (74,59) (74,53) (58,53)
        Rectangle (41,43 20x20), "P%d", text variable: mInst.nSelectedPoint
    RoundedRectangle (102,479 60x20), "Test", invisible if: mInst._bUT_4pPuc
        toggle mInst._bUT_4pPuc
END_VISUALIZATION

// ---- POUs/Print/DefGrid/_VISU_Templates/_VISU_DropSpeedComp_Setup.TcVIS
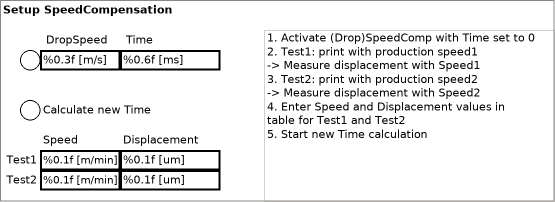
VISUALIZATION _VISU_DropSpeedComp_Setup  // 555x202
VAR_IN_OUT
	mInst : FB_DropSpeedComp;
END_VAR
    Rectangle (0,0 555x202)
    Ellipse (20,50 20x20), tooltip "Enable Correction"
        toggle mInst.bEnable p2164770859=TRUE
    Rectangle (40,50 80x20), "%0.3f [m/s]", tooltip "DropSpeed", text variable: mInst.fDropSpeed
        OnMouseClick: write the text variable via Default
    Rectangle (120,50 100x20), "%0.6f [ms]", tooltip "Dead/Add Time", text variable: mInst.fDropSpeedDeadTime
        OnMouseClick: write the text variable via Default
    Rectangle (123,30 78x20), "Time"
    Rectangle (43,30 78x20), "DropSpeed"
    Ellipse (20,100 20x20), tooltip "Calculate new time"
        tap mInst.bCalcDeadTime
    Rectangle (40,150 80x20), "%0.1f [m/min]", text variable: mInst.fTestSpeed[1], colour toggle: mInst.fTestSpeed[1] = 0
        OnMouseClick: write the text variable via Default
    Rectangle (40,170 80x20), "%0.1f [m/min]", text variable: mInst.fTestSpeed[2], colour toggle: mInst.fTestSpeed[2] = 0
        OnMouseClick: write the text variable via Default
    Rectangle (40,130 78x20), "Speed"
    Rectangle (120,150 100x20), "%0.1f [um]", text variable: mInst.fTestDisplacement[1]
        OnMouseClick: write the text variable via Default
    Rectangle (120,170 100x20), "%0.1f [um]", text variable: mInst.fTestDisplacement[2]
        OnMouseClick: write the text variable via Default
    Rectangle (120,130 100x20), "Displacement"
    Rectangle (0,0 256x20), "Setup SpeedCompensation"
    Rectangle (40,100 150x20), "Calculate new Time"
    Rectangle (0,150 40x20), "Test1"
    Rectangle (0,170 40x20), "Test2"
    Textfield (264,30 291x172), "1. Activate (Drop)SpeedComp with Time set to 0 2. Test1: print with production speed1 -> Measure displacement with Speed1 3. Test2: print with production speed2 -> Measure displacement with Speed2 4. Enter Speed and Displacement values in table for Test1 and Test2 5. Start new Time calculation"
END_VISUALIZATION

// ---- POUs/Print/DefGrid/_VISU_Templates/_VISU_CTGridExporter.TcVIS
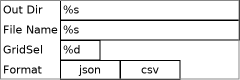
VISUALIZATION _VISU_CTGridExporter  // 240x80
VAR_IN_OUT
		mInst : FB_GridDataExporter;
END_VAR
    Rectangle (0,40 60x20), "GridSel"
    Rectangle (0,0 60x20), "Out Dir"
    Rectangle (0,60 60x20), "Format"
    RoundedRectangle (60,60 60x20), "json", colour toggle: mInst.sFileFormat = 'json'
        OnMouseClick: execute { mInst.sFileFormat := 'json'; }
    RoundedRectangle (120,60 60x20), "csv", colour toggle: mInst.sFileFormat = 'csv'
        OnMouseClick: execute { mInst.sFileFormat := 'csv'; }
    Rectangle (0,20 60x20), "File Name"
    Rectangle (60,40 40x20), "%d", text variable: mInst.nSelectGrid
        OnMouseClick: write the text variable via Default
    Rectangle (60,0 180x20), "%s", tooltip "%s", text variable: mInst.sOutputDir
        p4168582468: mInst.sOutputDir
        OnMouseClick: write the text variable via Default
    Rectangle (60,20 180x20), "%s", tooltip "%s", text variable: mInst.sFileName
        p4168582468: mInst.sFileName
        OnMouseClick: write the text variable via Default
END_VISUALIZATION

// ---- POUs/Print/Maxliner/_VISU_PmEnable_Maxliner.TcVIS
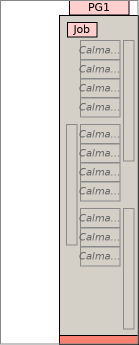
VISUALIZATION _VISU_PmEnable_Maxliner  // 139x345
VAR_IN_OUT
  mInst : FB_PrintModule_Maxliner;
END_VAR
    RoundedRectangle (59,15 80x329), tooltip "WorkerPrint enable"
        toggle mInst.fbWorkerPrint[1]._bEnable
    RoundedRectangle (69,0 60x15), "PG1", tooltip "PG enable"
        toggle mInst.fbWorkerPrint[1]._pAdsPg^.stAds.bI_Enable
    Frame (123,40 11x121)
        shows CalmarCompPrint._VISU_PC_MiniVertical(mInst := mInst._pPc[1]^)
    Frame (66,124 11x121)
        shows CalmarCompPrint._VISU_PC_MiniVertical(mInst := mInst._pPc[2]^)
    Frame (80,40 40x20)
        shows CalmarCompPrint._VISU_PH_TinyVertical(mInst := mInst._pPh[1]^)
    Frame (80,59 40x20)
        shows CalmarCompPrint._VISU_PH_TinyVertical(mInst := mInst._pPh[2]^)
    Frame (80,78 40x20)
        shows CalmarCompPrint._VISU_PH_TinyVertical(mInst := mInst._pPh[3]^)
    Frame (80,97 40x20)
        shows CalmarCompPrint._VISU_PH_TinyVertical(mInst := mInst._pPh[4]^)
    Frame (80,124 40x20)
        shows CalmarCompPrint._VISU_PH_TinyVertical(mInst := mInst._pPh[5]^)
    Frame (80,143 40x20)
        shows CalmarCompPrint._VISU_PH_TinyVertical(mInst := mInst._pPh[6]^)
    RoundedRectangle (67,22 30x15), "Job", tooltip "Job is active", colour toggle: mInst.fbWorkerPrint[1]._bJobActive
    RoundedRectangle (59,335 80x10), tooltip "Worker PrintEnable"
        toggle mInst.fbWorkerPrint[1].bWorkerPrintEnable
    Frame (80,162 40x20)
        shows CalmarCompPrint._VISU_PH_TinyVertical(mInst := mInst._pPh[7]^)
    Frame (80,181 40x20)
        shows CalmarCompPrint._VISU_PH_TinyVertical(mInst := mInst._pPh[8]^)
    Frame (123,208 11x121)
        shows CalmarCompPrint._VISU_PC_MiniVertical(mInst := mInst._pPc[3]^)
    Frame (80,208 40x20)
        shows CalmarCompPrint._VISU_PH_TinyVertical(mInst := mInst._pPh[9]^)
    Frame (80,227 40x20)
        shows CalmarCompPrint._VISU_PH_TinyVertical(mInst := mInst._pPh[10]^)
    Frame (80,246 40x20)
        shows CalmarCompPrint._VISU_PH_TinyVertical(mInst := mInst._pPh[11]^)
END_VISUALIZATION

// ---- POUs/Print/Maxliner/_VISU_Pm_Maxliner_ImgLengthCheck.TcVIS
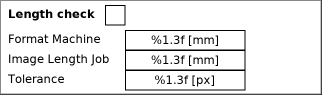
VISUALIZATION _VISU_Pm_Maxliner_ImgLengthCheck  // 322x95
VAR_IN_OUT
	mInst : FB_PrintModule_Maxliner;
END_VAR
    Rectangle (0,0 322x95)
    Rectangle (5,30 120x18), "Format Machine"
    Rectangle (5,5 96x18), "Length check"
    Rectangle (125,30 120x20), "%1.3f [mm]", text variable: mInst._pModuleMachineState^.fSubstrateLen * 1000
    Rectangle (5,50 120x18), "Image Length Job"
    Rectangle (125,50 120x20), "%1.3f [mm]", text variable: mInst.fbWorkerPrint[1]._fCurrentImgDepth * 1000
    RoundedRectangle (105,5 20x20), colour toggle: mInst._pModuleMachineFeedback^.bLengthMismatch
    Rectangle (5,70 120x18), "Tolerance"
    Rectangle (125,70 120x20), "%1.3f [px]", text variable: mInst.fC_FormatLengthTolerance
END_VISUALIZATION

// ---- POUs/Print/Maxliner/_VISU_Pm_Maxliner_Worker.TcVIS
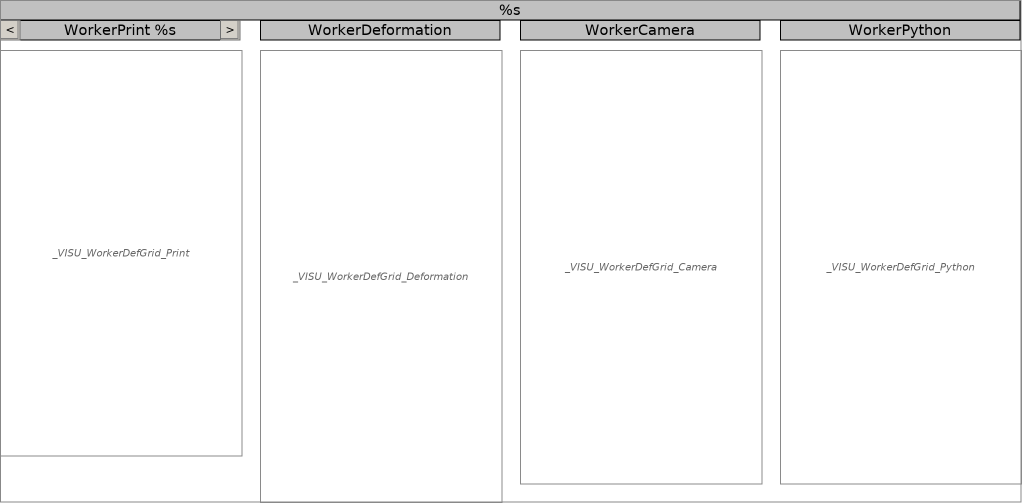
VISUALIZATION _VISU_Pm_Maxliner_Worker  // 1022x503
VAR_IN_OUT
	mInst : FB_PrintModule_Maxliner;
END_VAR
    Frame (0,50 242x406)
        shows _VISU_WorkerDefGrid_Print(m_Inst := mInst.fbWorkerPrint[mInst.fbView.nSelWorkerPrint])
    Rectangle (0,20 240x20), "WorkerPrint %s", text variable: mInst.fbView.nSelWorkerPrint
    Frame (520,50 242x434)
        shows _VISU_WorkerDefGrid_Camera(m_Inst := mInst.fbWorkerCamera)
    Rectangle (520,20 240x20), "WorkerCamera"
    Rectangle (0,0 1020x20), "%s", text variable: mInst.fbAdsPm.aO_Name
    Rectangle (260,20 240x20), "WorkerDeformation"
    Frame (260,50 242x453)
        shows _VISU_WorkerDefGrid_Deformation(m_Inst := mInst.fbWorkerDeformation)
    Button (0,20 20x20), "<"
        OnMouseClick: execute { mInst.fbView.nSelWorkerPrint := mInst.fbView.nSelWorkerPrint - 1; }
    Button (220,20 20x20), ">"
        OnMouseClick: execute { mInst.fbView.nSelWorkerPrint := mInst.fbView.nSelWorkerPrint + 1; }
    Rectangle (780,20 240x20), "WorkerPython"
    Frame (780,50 242x434)
        shows _VISU_WorkerDefGrid_Python(m_Inst := mInst.fbWorkerPython)
END_VISUALIZATION

// ---- POUs/Print/Maxliner/_VISU_Pm_Maxliner_mini_Worker.TcVIS
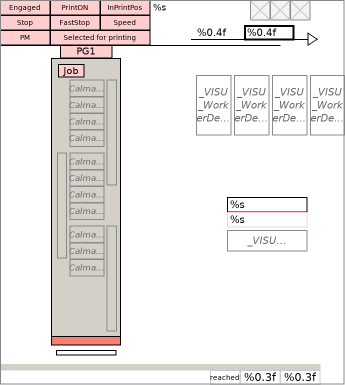
VISUALIZATION _VISU_Pm_Maxliner_mini_Worker  // 345x385
VAR_IN_OUT
  mInst : FB_PrintModule_Maxliner;
END_VAR
    Rectangle (150,0 160x15), "%s", text variable: mInst.fbAdsPm.stAds.aO_Name
    Rectangle (0,40 320x280)
    Frame (227,230 80x21)
        shows _VISU_MarkDetection_Trigger(mInst := mInst.fbMarkDetection)
    Rectangle (227,197 80x15), "%s", tooltip "active camera device", text variable: mInst.fbWorkerCamera._iActiveCam.sName
    Rectangle (227,212 80x15), "%s", tooltip "active camera mode", text variable: mInst.fbWorkerCamera._iActiveCam.eCameraMode, colour toggle: mInst.fbWorkerCamera._bCamValid
    RoundedRectangle (0,364 320x6), colour toggle: mInst.fbView.bMovingInd
    Frame (0,45 162x300)
        shows _VISU_PmEnable_Maxliner(mInst := mInst)
        p2738717112: mInst.fbView.zPos_PM
    RoundedRectangle (56,350 60x5), colour toggle: mInst.fbView.bPrintInd[1]
        p2738717112: mInst.fbView.zPos_PM
    Line (0,45) (280,45)
    RoundedRectangle (280,370 40x15), "%0.3f", tooltip "Target speed", text variable: mInst._pModuleMachineState^.fTargetSpeed
    RoundedRectangle (240,370 40x15), "%0.3f", tooltip "Current Speed", text variable: mInst.fSpeed
    RoundedRectangle (0,0 50x15), "Engaged", colour toggle: mInst._pModuleMachineState^.bEngaged
    RoundedRectangle (50,0 50x15), "PrintON", colour toggle: mInst._pModuleMachineState^.bPrintActivated
    RoundedRectangle (100,0 50x15), "InPrintPos", colour toggle: mInst._pModuleMachineState^.bUnitInPrintPosition
    RoundedRectangle (0,15 50x15), "Stop", colour toggle: NOT mInst._pModuleMachineState^.bStopRequest
    RoundedRectangle (50,15 50x15), "FastStop", colour toggle: NOT mInst._pModuleMachineState^.bFastStopRequest
    RoundedRectangle (100,15 50x15), "Speed", colour toggle: mInst.bSpeedReachedForPrinting
    Image (250,0 20x20), invisible if: NOT mInst._pModuleMachineState^.bSleep, image: ImagePool_Steinemann.sleep_icon
    Image (270,0 20x20), invisible if: NOT mInst._pModuleMachineState^.bShutdown, image: ImagePool_Steinemann.shutdown_icon
    Image (290,0 20x20), invisible if: NOT mInst._pModuleMachineState^.bEStop, image: ImagePool_Steinemann.estop_icon
    RoundedRectangle (210,370 30x15), "reached", tooltip "Target speed reached", colour toggle: mInst._pModuleMachineState^.bTargetSpeedReached
    Frame (234,75 35x60)
        shows _VISU_WorkerDefGrid_small(m_Inst := mInst.fbWorkerDeformation)
    Frame (272,75 35x60)
        shows _VISU_WorkerDefGrid_small(m_Inst := mInst.fbWorkerCamera)
    Frame (196,75 35x60)
        shows _VISU_WorkerDefGrid_small(m_Inst := mInst.fbWorkerPrint[1])
    RoundedRectangle (50,30 100x15), "Selected for printing"
        toggle mInst.bSelectedForPrint
    RoundedRectangle (0,30 50x15), "PM"
        toggle mInst.fbAdsPm.stAds.bI_Enable
    Rectangle (194,25 50x15), "%0.4f", tooltip "PM position on main tracker", text variable: mInst._fPmMainTrackPos
    Polyline (191,39) (308,39) (308,33) (317,39) (308,45) (308,39)
    Rectangle (244,25 50x15), "%0.4f", tooltip "PM position to previous", text variable: mInst._fPmDistToPrev
        OnMouseClick: write the text variable via Default
    Frame (310,75 35x60)
        shows _VISU_WorkerDefGrid_small(m_Inst := mInst.fbWorkerPython)
END_VISUALIZATION

// ---- POUs/Print/Maxliner/_VISU_Pm_Maxliner_Debug.TcVIS
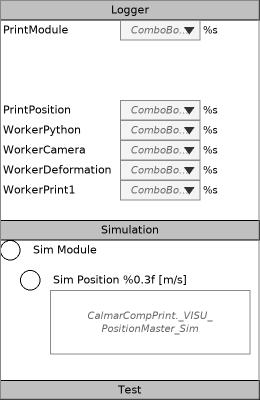
VISUALIZATION _VISU_Pm_Maxliner_Debug  // 260x400
VAR_IN_OUT
	mInst : FB_PrintModule_Maxliner;
END_VAR
    Rectangle (0,220 260x20), "Simulation"
    Ellipse (20,270 20x20), tooltip "Sim position"
        toggle mInst.fbPrintPosition._bSim
    Rectangle (50,270 200x20), "Sim Position %0.3f [m/s]", text variable: mInst.fbPrintPosition.fbPositionMaster._fSimSpeed
        OnMouseClick: write the text variable via Default
    Rectangle (0,0 260x20), "Logger"
    Rectangle (0,100 120x20), "PrintPosition"
    Rectangle (200,100 60x20), "%s", tooltip "LogLevel", text variable: mInst.fbPrintPosition._loglevel
        OnMouseClick: write the text variable via Default
    Rectangle (0,140 120x20), "WorkerCamera"
    Rectangle (200,140 60x20), "%s", tooltip "LogLevel", text variable: mInst.fbWorkerCamera._loglevel
        OnMouseClick: write the text variable via Default
    Rectangle (0,180 120x20), "WorkerPrint1"
    Rectangle (200,180 60x20), "%s", tooltip "LogLevel", text variable: mInst.fbWorkerPrint[1]._loglevel
        OnMouseClick: write the text variable via Default
    Rectangle (0,160 120x20), "WorkerDeformation"
    Rectangle (200,160 60x20), "%s", tooltip "LogLevel", text variable: mInst.fbWorkerDeformation._loglevel
        OnMouseClick: write the text variable via Default
    ComboBoxInteger (120,180 80x20), tooltip "LogLevel", variable: mInst.fbWorkerPrint[1]._loglevel, text list: 'LogSeverity'
    ComboBoxInteger (120,160 80x20), tooltip "LogLevel", variable: mInst.fbWorkerDeformation._loglevel, text list: 'LogSeverity'
    ComboBoxInteger (120,140 80x20), tooltip "LogLevel", variable: mInst.fbWorkerCamera._loglevel, text list: 'LogSeverity'
    ComboBoxInteger (120,100 80x20), tooltip "LogLevel", variable: mInst.fbPrintPosition._loglevel, text list: 'LogSeverity'
    Frame (50,290 200x64)
        shows CalmarCompPrint._VISU_PositionMaster_Sim(mInst := mInst.fbPrintPosition.fbPositionMaster)
    Rectangle (0,380 260x20), "Test"
    Ellipse (0,240 20x20), tooltip "Sim position"
        toggle mInst.bSimEnable
    Rectangle (30,240 200x20), "Sim Module"
    Rectangle (0,20 120x20), "PrintModule"
    Rectangle (200,20 60x20), "%s", tooltip "LogLevel", text variable: mInst._loglevel
        OnMouseClick: write the text variable via Default
    ComboBoxInteger (120,20 80x20), tooltip "LogLevel", variable: mInst._loglevel, text list: 'LogSeverity'
    Rectangle (0,120 120x20), "WorkerPython"
    Rectangle (200,120 60x20), "%s", tooltip "LogLevel", text variable: mInst.fbWorkerPython._loglevel
        OnMouseClick: write the text variable via Default
    ComboBoxInteger (120,120 80x20), tooltip "LogLevel", variable: mInst.fbWorkerPython._loglevel, text list: 'LogSeverity'
END_VISUALIZATION

// ---- POUs/Print/Maxliner/_VISU_Pm_Maxliner.TcVIS
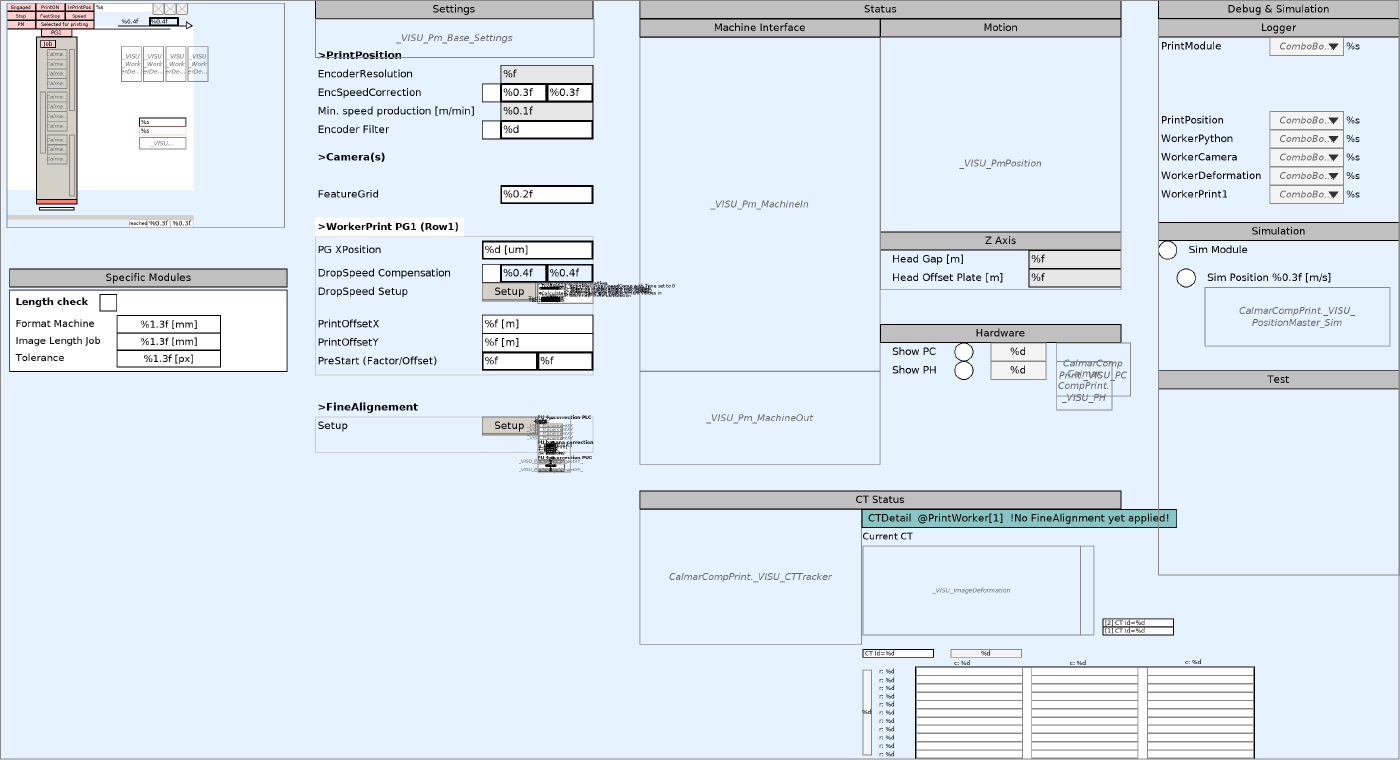
VISUALIZATION _VISU_Pm_Maxliner  // 1511x821
VAR_IN_OUT
  mInst : FB_PrintModule_Maxliner;
END_VAR
    Frame (10,313 300x90)
        shows _VISU_Pm_Maxliner_ImgLengthCheck(mInst := mInst)
    Frame (690,550 240x146)
        shows CalmarCompPrint._VISU_CTTracker(mInst := mInst.fbCTTracker)
    Frame (931,570 428x251)
        shows _VISU_CT_Details(mInst := mInst.fbWorkerPrint[1])
    Rectangle (930,550 340x20), "CTDetail @PrintWorker[1] !No FineAlignment yet applied!"
    Rectangle (690,530 520x20), "CT Status"
    Frame (690,401 260x101)
        shows _VISU_Pm_MachineOut(ref := mInst._pModuleMachineFeedback^)
    Frame (690,40 260x361)
        shows _VISU_Pm_MachineIn(ref := mInst._pModuleMachineState^)
    Rectangle (690,20 260x20), "Machine Interface"
    Rectangle (950,20 260x20), "Motion"
    Frame (7,3 300x243)
        shows _VISU_Pm_Maxliner_mini_Worker(mInst := mInst)
    Rectangle (950,350 260x20), "Hardware"
    Frame (1250,20 261x601), invisible if: NOT mInst.fbView.bShowDebugAndSim
        shows _VISU_Pm_Maxliner_Debug(mInst := mInst)
    Rectangle (340,0 300x20), "Settings"
    Rectangle (690,0 520x20), "Status"
    Rectangle (1250,0 260x20), "Debug & Simulation"
        toggle mInst.fbView.bShowDebugAndSim
    Rectangle (950,250 260x20), "Z Axis"
    Rectangle (960,270 140x20), "Head Gap [m]"
    Rectangle (1110,270 100x20), "%f", text variable: mInst._pModuleMachineFeedback^.fHeadGap
    Rectangle (960,290 140x20), "Head Offset Plate [m]"
    Rectangle (1110,290 100x20), "%f", text variable: mInst.fC_HeadOffsetPlate
    Frame (1140,370 80x58), invisible if: NOT mInst.fbView.bShowPcDetail
        shows CalmarCompPrint._VISU_PC(mInst := mInst._pPc[mInst.fbView.nSelPcDetail]^)
    Rectangle (960,390 110x20), "Show PH"
    Rectangle (960,370 110x20), "Show PC"
    Ellipse (1030,390 20x20)
        toggle mInst.fbView.bShowPhDetail
    Ellipse (1030,370 20x20)
        toggle mInst.fbView.bShowPcDetail
    Frame (1140,390 60x53), invisible if: NOT mInst.fbView.bShowPhDetail
        shows CalmarCompPrint._VISU_PH(mInst := mInst._pPh[mInst.fbView.nSelPhDetail]^)
    Scrollbar (1069,390 60x20), "%d", text variable: mInst.fbView.nSelPhDetail, invisible if: NOT mInst.fbView.bShowPhDetail
        p2245068023: mInst._nPh
        p1057716461: mInst.fbView.nSelPhDetail
    Scrollbar (1069,370 60x20), "%d", text variable: mInst.fbView.nSelPcDetail, invisible if: NOT mInst.fbView.bShowPcDetail
        p2245068023: mInst._nPc
        p1057716461: mInst.fbView.nSelPcDetail
    Rectangle (10,290 300x20), "Specific Modules"
    Frame (340,20 299x522)
        shows _VISU_Pm_Maxliner_Settings(mInst := mInst)
        p4053072137: mInst
    Frame (950,40 260x273)
        shows _VISU_PmPosition(mInst := mInst)
END_VISUALIZATION

// ---- POUs/Print/Maxliner/_VISU_Pm_Maxliner_Settings.TcVIS
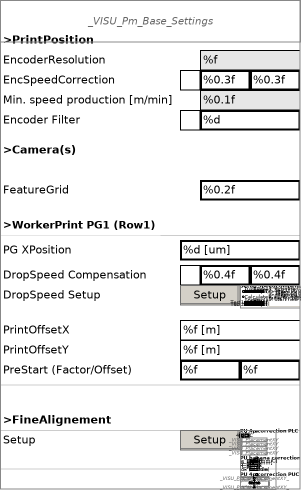
VISUALIZATION _VISU_Pm_Maxliner_Settings  // 301x490
VAR_IN_OUT
	mInst : FB_PrintModule_Maxliner;
END_VAR
    Rectangle (0,430 300x39)
    Rectangle (250,70 50x20), "%0.3f", tooltip "Encoder speed compensation reference speed", text variable: mInst.fbPrintPosition._fSpeedCompRefSpeed
        OnMouseClick: write the text variable via Default
    Rectangle (200,70 50x20), "%0.3f", tooltip "Encoder speed compensation factor", text variable: mInst.fbPrintPosition._fSpeedCompFactor
        OnMouseClick: write the text variable via Default
    RoundedRectangle (180,70 20x20)
        toggle mInst.fbPrintPosition._bEnSpeedComp
    Rectangle (0,70 180x20), "EncSpeedCorrection"
    Rectangle (0,50 180x20), "EncoderResolution"
    Rectangle (200,50 100x20), "%f", tooltip "by calculation", text variable: mInst.fbPrintPosition._fEncoderResolution
    Rectangle (0,235 300x150)
    Rectangle (0,265 180x20), "DropSpeed Compensation"
    Rectangle (200,265 50x20), "%0.4f", tooltip "DropSpeed [m/s]", text variable: mInst.fbWorkerPrint[1].fbDropSpeedComp.fDropSpeed
        OnMouseClick: write the text variable via Default
    Rectangle (250,265 50x20), "%0.4f", tooltip "Dead/Add Time [ms]", text variable: mInst.fbWorkerPrint[1].fbDropSpeedComp.fDropSpeedDeadTime
        OnMouseClick: write the text variable via Default
    RoundedRectangle (180,265 20x20), tooltip "Enabled compensation", input disabled if: TRUE
        toggle mInst.fbWorkerPrint[1].fbDropSpeedComp._bEnable p2164770859=TRUE
    Button (180,285 60x20), "Setup", tooltip "Setup"
        toggle mInst.fbWorkerPrint[1].bShowDropSpeedSetup
    Rectangle (0,285 180x20), "DropSpeed Setup"
    Rectangle (0,30 180x20), ">PrintPosition"
    Rectangle (0,90 180x20), "Min. speed production [m/min]"
    Rectangle (200,90 100x20), "%0.1f", tooltip "constant", text variable: mInst.fC_MinimalProductionSpeed_in_MpMin
    Rectangle (0,140 180x20), ">Camera(s)"
    Rectangle (200,110 100x20), "%d", tooltip "Filter depth", text variable: mInst.fbPrintPosition.fbPositionMaster.nFilterDepth
        OnMouseClick: write the text variable via Default
    RoundedRectangle (180,110 20x20)
        toggle mInst.fbPrintPosition.fbPositionMaster.bEnableFilter
    Rectangle (0,110 180x20), "Encoder Filter"
    Rectangle (0,180 180x20), "FeatureGrid"
    Rectangle (200,180 100x20), "%0.2f", text variable: mInst.fbWorkerCamera._fFeatureGrid
        OnMouseDown: write the text variable via Default
    Rectangle (0,410 180x20), ">FineAlignement"
    Button (180,430 60x20), "Setup", tooltip "Setup"
        toggle minst.fbView.bShowFineAlignement
    Rectangle (0,430 180x20), "Setup"
    Frame (0,0 301x42)
        shows _VISU_Pm_Base_Settings(mInst := mInst)
    Rectangle (0,320 180x20), "PrintOffsetX"
    Rectangle (0,340 180x20), "PrintOffsetY"
    Rectangle (180,320 120x20), "%f [m]", text variable: mInst.fbWorkerPrint[1].fPrintStartOffset, input disabled if: TRUE
    Rectangle (180,340 120x20), "%f [m]", text variable: mInst.fbWorkerPrint[1].fPrintYOffset, input disabled if: TRUE
    Rectangle (0,215 160x20), ">WorkerPrint PG1 (Row1)"
    Rectangle (0,240 180x20), "PG XPosition"
    Rectangle (180,240 120x20), "%d [um]", text variable: mInst.fbAdsPg[1].stAds.sI_ShiftPositionX.lI_Val
        OnMouseClick: write the text variable via Default
    Rectangle (0,360 180x20), "PreStart (Factor/Offset)"
    Rectangle (180,360 60x20), "%f", tooltip "PreStart ShiftFactor", text variable: mInst.fbWorkerPrint[1]._fStartShiftFactor
        OnMouseClick: write the text variable via Default
    Rectangle (240,360 60x20), "%f", tooltip "PreStart ShiftOffset", text variable: mInst.fbWorkerPrint[1]._fStartShiftOffset
        OnMouseClick: write the text variable via Default
    Frame (240,285 60x23), invisible if: NOT mInst.fbWorkerPrint[1].bShowDropSpeedSetup
        shows _VISU_DropSpeedComp_Setup(mInst := mInst.fbWorkerPrint[1].fbDropSpeedComp)
    Frame (240,430 36x60), invisible if: NOT minst.fbView.bShowFineAlignement
        shows _VISU_FineAlignment(mInst := mInst.fbFineAlignement)
END_VISUALIZATION

// ---- POUs/Print/WEU/_VISU_PmImgLengthCheck.TcVIS
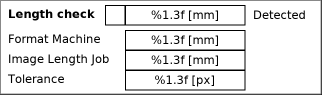
VISUALIZATION _VISU_PmImgLengthCheck  // 322x95
VAR_IN_OUT
	mInst : FB_PrintModule_WEU;
END_VAR
    Rectangle (0,0 322x95)
    Rectangle (5,30 120x18), "Format Machine"
    Rectangle (5,5 96x18), "Length check"
    Rectangle (125,30 120x20), "%1.3f [mm]", text variable: mInst._pModuleMachineState^.fSubstrateLen * 1000
    Rectangle (5,50 120x18), "Image Length Job"
    Rectangle (125,50 120x20), "%1.3f [mm]", text variable: mInst.fbWorkerPrint[1]._fCurrentImgDepth * 1000
    RoundedRectangle (105,5 20x20), colour toggle: mInst._pModuleMachineFeedback^.bLengthMismatch
    Rectangle (5,70 120x18), "Tolerance"
    Rectangle (125,70 120x20), "%1.3f [px]", text variable: mInst.fC_FormatLengthTolerance
    Rectangle (250,6 60x18), "Detected"
    Rectangle (125,5 120x20), "%1.3f [mm]", text variable: mInst.fbMarkCameraWeu.fbMarkDetection._fImageLengthEffective * 1000
END_VISUALIZATION

// ---- POUs/Print/WEU/_VISU_Pm_WEU_Debug.TcVIS
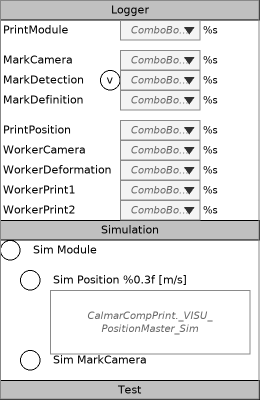
VISUALIZATION _VISU_Pm_WEU_Debug  // 260x400
VAR_IN_OUT
	mInst : FB_PrintModule_WEU;
END_VAR
    Rectangle (0,220 260x20), "Simulation"
    Ellipse (20,270 20x20), tooltip "Sim position"
        toggle mInst.fbPrintPosition._bSim
    Rectangle (50,270 200x20), "Sim Position %0.3f [m/s]", text variable: mInst.fbPrintPosition.fbPositionMaster._fSimSpeed
        OnMouseClick: write the text variable via Default
    Ellipse (20,350 20x20)
        toggle mInst.fbMarkCameraWeu.bSimulate
    Rectangle (50,350 200x20), "Sim MarkCamera"
    Rectangle (0,0 260x20), "Logger"
    Rectangle (0,70 120x20), "MarkDetection"
    Rectangle (0,90 120x20), "MarkDefinition"
    Rectangle (200,90 60x20), "%s", tooltip "LogLevel", text variable: mInst.fbMarkCameraWeu.fbMarkDefinition._loglevel
        OnMouseClick: write the text variable via Default
    Rectangle (0,50 120x20), "MarkCamera"
    Rectangle (200,50 60x20), "%s", tooltip "LogLevel", text variable: mInst.fbMarkCameraWeu._loglevel
        OnMouseClick: write the text variable via Default
    Rectangle (0,120 120x20), "PrintPosition"
    Rectangle (200,120 60x20), "%s", tooltip "LogLevel", text variable: mInst.fbPrintPosition._loglevel
        OnMouseClick: write the text variable via Default
    Rectangle (0,140 120x20), "WorkerCamera"
    Rectangle (200,140 60x20), "%s", tooltip "LogLevel", text variable: mInst.fbWorkerCamera._loglevel
        OnMouseClick: write the text variable via Default
    Rectangle (0,180 120x20), "WorkerPrint1"
    Rectangle (200,180 60x20), "%s", tooltip "LogLevel", text variable: mInst.fbWorkerPrint[1]._loglevel
        OnMouseClick: write the text variable via Default
    Ellipse (100,70 20x20), "v", tooltip "Verbose mode"
        toggle mInst.fbMarkCameraWeu.fbMarkDetection._bVerbose
    Rectangle (0,160 120x20), "WorkerDeformation"
    Rectangle (200,160 60x20), "%s", tooltip "LogLevel", text variable: mInst.fbWorkerDeformation._loglevel
        OnMouseClick: write the text variable via Default
    ComboBoxInteger (120,180 80x20), tooltip "LogLevel", variable: mInst.fbWorkerPrint[1]._loglevel, text list: 'LogSeverity'
    ComboBoxInteger (120,160 80x20), tooltip "LogLevel", variable: mInst.fbWorkerDeformation._loglevel, text list: 'LogSeverity'
    ComboBoxInteger (120,140 80x20), tooltip "LogLevel", variable: mInst.fbWorkerCamera._loglevel, text list: 'LogSeverity'
    ComboBoxInteger (120,120 80x20), tooltip "LogLevel", variable: mInst.fbPrintPosition._loglevel, text list: 'LogSeverity'
    ComboBoxInteger (120,50 80x20), tooltip "LogLevel", variable: mInst.fbMarkCameraWeu._loglevel, text list: 'LogSeverity'
    ComboBoxInteger (120,90 80x20), tooltip "LogLevel", variable: mInst.fbMarkCameraWeu.fbMarkDefinition._loglevel, text list: 'LogSeverity'
    Rectangle (200,70 60x20), "%s", tooltip "LogLevel", text variable: mInst.fbMarkCameraWeu.fbMarkDetection._loglevel
        OnMouseClick: write the text variable via Default
    ComboBoxInteger (120,70 80x20), tooltip "LogLevel", variable: mInst.fbMarkCameraWeu.fbMarkDetection._loglevel, text list: 'LogSeverity'
    Frame (50,290 200x64)
        shows CalmarCompPrint._VISU_PositionMaster_Sim(mInst := mInst.fbPrintPosition.fbPositionMaster)
    Rectangle (0,380 260x20), "Test"
    Ellipse (0,240 20x20), tooltip "Sim position"
        toggle mInst.bSimEnable
    Rectangle (30,240 200x20), "Sim Module"
    Rectangle (0,20 120x20), "PrintModule"
    Rectangle (200,20 60x20), "%s", tooltip "LogLevel", text variable: mInst._loglevel
        OnMouseClick: write the text variable via Default
    ComboBoxInteger (120,20 80x20), tooltip "LogLevel", variable: mInst._loglevel, text list: 'LogSeverity'
    Rectangle (0,200 120x20), "WorkerPrint2"
    Rectangle (200,200 60x20), "%s", tooltip "LogLevel", text variable: mInst.fbWorkerPrint[2]._loglevel
        OnMouseClick: write the text variable via Default
    ComboBoxInteger (120,200 80x20), tooltip "LogLevel", variable: mInst.fbWorkerPrint[2]._loglevel, text list: 'LogSeverity'
END_VISUALIZATION

// ---- POUs/Print/WEU/_VISU_Pm_WEU_Settings.TcVIS
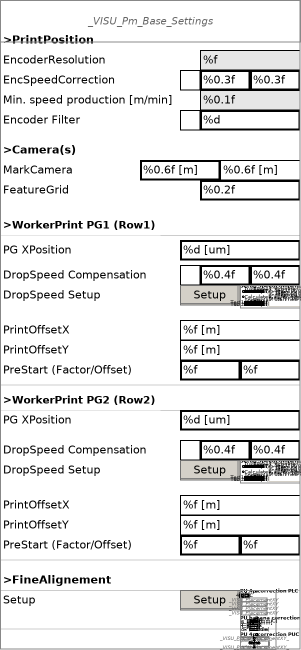
VISUALIZATION _VISU_Pm_WEU_Settings  // 301x650
VAR_IN_OUT
	mInst : FB_PrintModule_WEU;
END_VAR
    Rectangle (0,590 300x39)
    Rectangle (250,70 50x20), "%0.3f", tooltip "Encoder speed compensation reference speed", text variable: mInst.fbPrintPosition._fSpeedCompRefSpeed
        OnMouseClick: write the text variable via Default
    Rectangle (200,70 50x20), "%0.3f", tooltip "Encoder speed compensation factor", text variable: mInst.fbPrintPosition._fSpeedCompFactor
        OnMouseClick: write the text variable via Default
    RoundedRectangle (180,70 20x20)
        toggle mInst.fbPrintPosition._bEnSpeedComp
    Rectangle (0,70 180x20), "EncSpeedCorrection"
    Rectangle (0,50 180x20), "EncoderResolution"
    Rectangle (200,50 100x20), "%f", tooltip "by calculation", text variable: mInst.fbPrintPosition._fEncoderResolution
    Rectangle (0,235 300x150)
    Rectangle (0,265 180x20), "DropSpeed Compensation"
    Rectangle (200,265 50x20), "%0.4f", tooltip "DropSpeed [m/s]", text variable: mInst.fbWorkerPrint[1].fbDropSpeedComp.fDropSpeed
        OnMouseClick: write the text variable via Default
    Rectangle (250,265 50x20), "%0.4f", tooltip "Dead/Add Time [ms]", text variable: mInst.fbWorkerPrint[1].fbDropSpeedComp.fDropSpeedDeadTime
        OnMouseClick: write the text variable via Default
    RoundedRectangle (180,265 20x20), tooltip "Enabled compensation", input disabled if: TRUE
        toggle mInst.fbWorkerPrint[1].fbDropSpeedComp._bEnable p2164770859=TRUE
    Button (180,285 60x20), "Setup", tooltip "Setup"
        toggle mInst.fbWorkerPrint[1].bShowDropSpeedSetup
    Rectangle (0,285 180x20), "DropSpeed Setup"
    Rectangle (0,30 180x20), ">PrintPosition"
    Rectangle (0,90 180x20), "Min. speed production [m/min]"
    Rectangle (200,90 100x20), "%0.1f", tooltip "constant", text variable: mInst.fC_MinimalProductionSpeed_in_MpMin
    Rectangle (0,140 180x20), ">Camera(s)"
    Rectangle (220,160 80x20), "%0.6f [m]", tooltip "(not used) CameraToPrintUnit", text variable: mInst.fbMarkCameraWeu._fCameraToPrintOffset, input disabled if: TRUE
        OnMouseDown: write the text variable via Default
    Rectangle (140,160 80x20), "%0.6f [m]", tooltip "DetectToCamera", text variable: mInst.fbMarkCameraWeu._fDetectToCameraOffset
        OnMouseDown: write the text variable via Default
    Rectangle (0,160 140x20), "MarkCamera"
    Rectangle (200,110 100x20), "%d", tooltip "Filter depth", text variable: mInst.fbPrintPosition.fbPositionMaster.nFilterDepth
        OnMouseClick: write the text variable via Default
    RoundedRectangle (180,110 20x20)
        toggle mInst.fbPrintPosition.fbPositionMaster.bEnableFilter
    Rectangle (0,110 180x20), "Encoder Filter"
    Rectangle (0,180 180x20), "FeatureGrid"
    Rectangle (200,180 100x20), "%0.2f", text variable: mInst.fbWorkerCamera._fFeatureGrid
        OnMouseDown: write the text variable via Default
    Rectangle (0,570 180x20), ">FineAlignement"
    Button (180,590 60x20), "Setup", tooltip "Setup"
        toggle minst.fbView.bShowFineAlignement
    Rectangle (0,590 180x20), "Setup"
    Frame (0,0 301x42)
        shows _VISU_Pm_Base_Settings(mInst := mInst)
    Rectangle (0,320 180x20), "PrintOffsetX"
    Rectangle (0,340 180x20), "PrintOffsetY"
    Rectangle (180,320 120x20), "%f [m]", text variable: mInst.fbWorkerPrint[1].fPrintStartOffset, input disabled if: TRUE
    Rectangle (180,340 120x20), "%f [m]", text variable: mInst.fbWorkerPrint[1].fPrintYOffset, input disabled if: TRUE
    Rectangle (0,410 300x150)
    Rectangle (0,440 180x20), "DropSpeed Compensation"
    Rectangle (200,440 50x20), "%0.4f", tooltip "DropSpeed [m/s]", text variable: mInst.fbWorkerPrint[2].fbDropSpeedComp.fDropSpeed
        OnMouseClick: write the text variable via Default
    Rectangle (250,440 50x20), "%0.4f", tooltip "Dead/Add Time [ms]", text variable: mInst.fbWorkerPrint[2].fbDropSpeedComp.fDropSpeedDeadTime
        OnMouseClick: write the text variable via Default
    RoundedRectangle (180,440 20x20), tooltip "Enabled compensation", input disabled if: TRUE
        toggle mInst.fbWorkerPrint[2].fbDropSpeedComp._bEnable p2164770859=TRUE
    Button (180,460 60x20), "Setup", tooltip "Setup"
        toggle mInst.fbWorkerPrint[2].bShowDropSpeedSetup
    Rectangle (0,460 180x20), "DropSpeed Setup"
    Rectangle (0,495 180x20), "PrintOffsetX"
    Rectangle (0,515 180x20), "PrintOffsetY"
    Rectangle (180,495 120x20), "%f [m]", text variable: mInst.fbWorkerPrint[2].fPrintStartOffset, input disabled if: TRUE
    Rectangle (180,515 120x20), "%f [m]", text variable: mInst.fbWorkerPrint[2].fPrintYOffset, input disabled if: TRUE
    Rectangle (0,390 160x20), ">WorkerPrint PG2 (Row2)"
    Rectangle (0,215 160x20), ">WorkerPrint PG1 (Row1)"
    Rectangle (0,240 180x20), "PG XPosition"
    Rectangle (180,240 120x20), "%d [um]", text variable: mInst.fbAdsPg[1].stAds.sI_ShiftPositionX.lI_Val
        OnMouseClick: write the text variable via Default
    Rectangle (0,410 180x20), "PG XPosition"
    Rectangle (180,410 120x20), "%d [um]", text variable: mInst.fbAdsPg[2].stAds.sI_ShiftPositionX.lI_Val
        OnMouseClick: write the text variable via Default
    Rectangle (0,360 180x20), "PreStart (Factor/Offset)"
    Rectangle (180,360 60x20), "%f", tooltip "PreStart ShiftFactor", text variable: mInst.fbWorkerPrint[1]._fStartShiftFactor
        OnMouseClick: write the text variable via Default
    Rectangle (240,360 60x20), "%f", tooltip "PreStart ShiftOffset", text variable: mInst.fbWorkerPrint[1]._fStartShiftOffset
        OnMouseClick: write the text variable via Default
    Rectangle (0,535 180x20), "PreStart (Factor/Offset)"
    Rectangle (180,535 60x20), "%f", tooltip "PreStart ShiftFactor", text variable: mInst.fbWorkerPrint[2]._fStartShiftFactor
        OnMouseClick: write the text variable via Default
    Rectangle (240,535 60x20), "%f", tooltip "PreStart ShiftOffset", text variable: mInst.fbWorkerPrint[2]._fStartShiftOffset
        OnMouseClick: write the text variable via Default
    Frame (240,460 60x23), invisible if: NOT mInst.fbWorkerPrint[2].bShowDropSpeedSetup
        shows _VISU_DropSpeedComp_Setup(mInst := mInst.fbWorkerPrint[2].fbDropSpeedComp)
    Frame (240,285 60x23), invisible if: NOT mInst.fbWorkerPrint[1].bShowDropSpeedSetup
        shows _VISU_DropSpeedComp_Setup(mInst := mInst.fbWorkerPrint[1].fbDropSpeedComp)
    Frame (240,590 36x60), invisible if: NOT minst.fbView.bShowFineAlignement
        shows _VISU_FineAlignment(mInst := mInst.fbFineAlignement)
END_VISUALIZATION

// ---- POUs/Print/WEU/_VISU_Pm_WEU.TcVIS
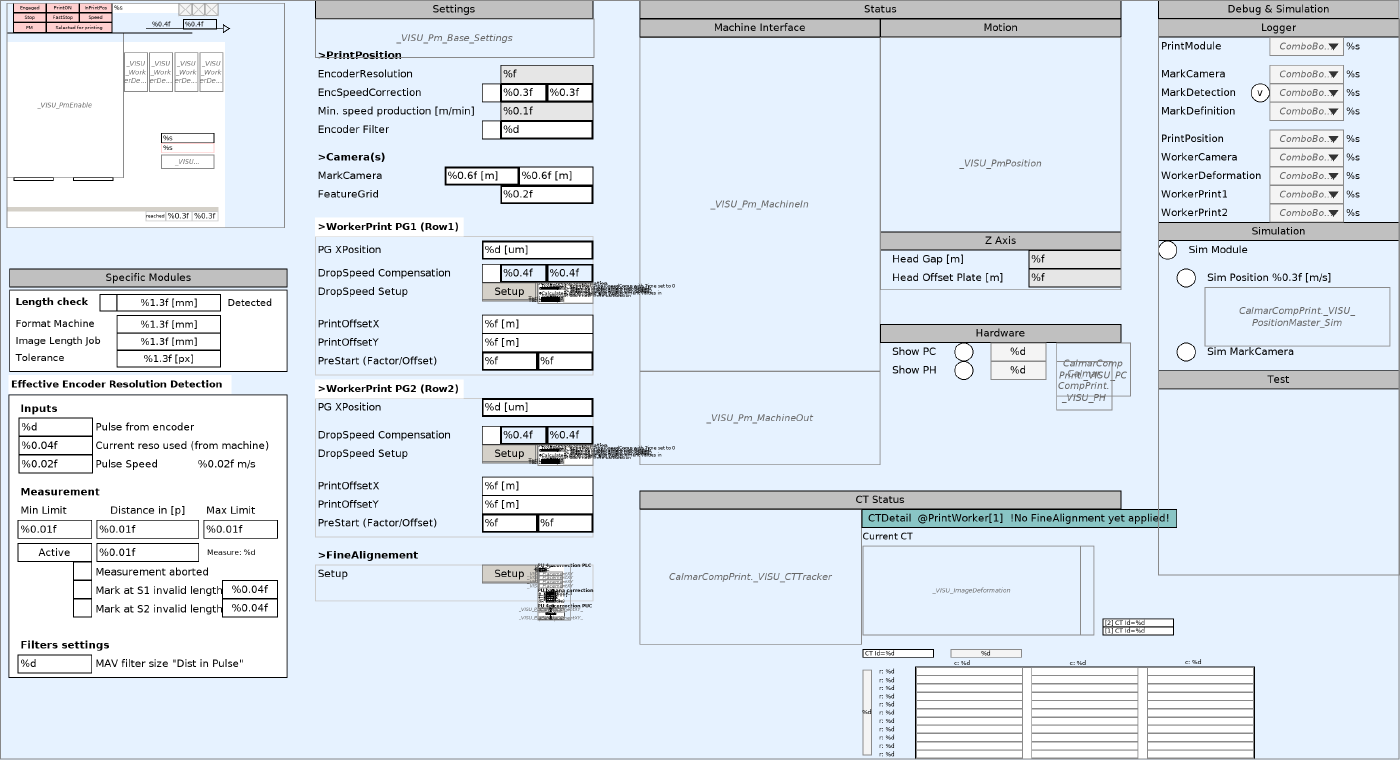
VISUALIZATION _VISU_Pm_WEU  // 1511x821
VAR_IN_OUT
  mInst : FB_PrintModule_WEU;
END_VAR
    Frame (10,313 300x90)
        shows _VISU_PmImgLengthCheck(mInst := mInst)
    Frame (690,550 240x146)
        shows CalmarCompPrint._VISU_CTTracker(mInst := mInst.fbCTTracker)
    Frame (931,570 428x251)
        shows _VISU_CT_Details(mInst := mInst.fbWorkerPrint[1])
    Rectangle (930,550 340x20), "CTDetail @PrintWorker[1] !No FineAlignment yet applied!"
    Rectangle (690,530 520x20), "CT Status"
    Frame (690,401 260x101)
        shows _VISU_Pm_MachineOut(ref := mInst._pModuleMachineFeedback^)
    Frame (690,40 260x361)
        shows _VISU_Pm_MachineIn(ref := mInst._pModuleMachineState^)
    Rectangle (690,20 260x20), "Machine Interface"
    Rectangle (950,20 260x20), "Motion"
    Frame (7,3 300x243)
        shows _VISU_Pm_WEU_mini(mInst := mInst)
    Rectangle (950,350 260x20), "Hardware"
    Frame (1250,20 261x601), invisible if: NOT mInst.fbView.bShowDebugAndSim
        shows _VISU_Pm_WEU_Debug(mInst := mInst)
    Rectangle (340,0 300x20), "Settings"
    Rectangle (690,0 520x20), "Status"
    Rectangle (1250,0 260x20), "Debug & Simulation"
        toggle mInst.fbView.bShowDebugAndSim
    Rectangle (950,250 260x20), "Z Axis"
    Rectangle (960,270 140x20), "Head Gap [m]"
    Rectangle (1110,270 100x20), "%f", text variable: mInst._pModuleMachineFeedback^.fHeadGap
    Rectangle (960,290 140x20), "Head Offset Plate [m]"
    Rectangle (1110,290 100x20), "%f", text variable: mInst.fC_HeadOffsetPlate
    Frame (1140,370 80x58), invisible if: NOT mInst.fbView.bShowPcDetail
        shows CalmarCompPrint._VISU_PC(mInst := mInst._pPc[mInst.fbView.nSelPcDetail]^)
    Rectangle (960,390 110x20), "Show PH"
    Rectangle (960,370 110x20), "Show PC"
    Ellipse (1030,390 20x20)
        toggle mInst.fbView.bShowPhDetail
    Ellipse (1030,370 20x20)
        toggle mInst.fbView.bShowPcDetail
    Frame (1140,390 60x53), invisible if: NOT mInst.fbView.bShowPhDetail
        shows CalmarCompPrint._VISU_PH(mInst := mInst._pPh[mInst.fbView.nSelPhDetail]^)
    Scrollbar (1069,390 60x20), "%d", text variable: mInst.fbView.nSelPhDetail, invisible if: NOT mInst.fbView.bShowPhDetail
        p2245068023: mInst._nPh
        p1057716461: mInst.fbView.nSelPhDetail
    Scrollbar (1069,370 60x20), "%d", text variable: mInst.fbView.nSelPcDetail, invisible if: NOT mInst.fbView.bShowPcDetail
        p2245068023: mInst._nPc
        p1057716461: mInst.fbView.nSelPcDetail
    Rectangle (10,290 300x20), "Specific Modules"
    Frame (9,405 301x362)
        shows _VISU_EffectiveEncoderResolutionDetection(mInst := mInst.fbEncoderResoDetect)
    Frame (340,20 299x522)
        shows _VISU_Pm_WEU_Settings(mInst := mInst)
    Frame (950,40 260x273)
        shows _VISU_PmPosition(mInst := mInst)
END_VISUALIZATION

// ---- POUs/Print/WEU/_VISU_Pm_WEU_1Worker.TcVIS
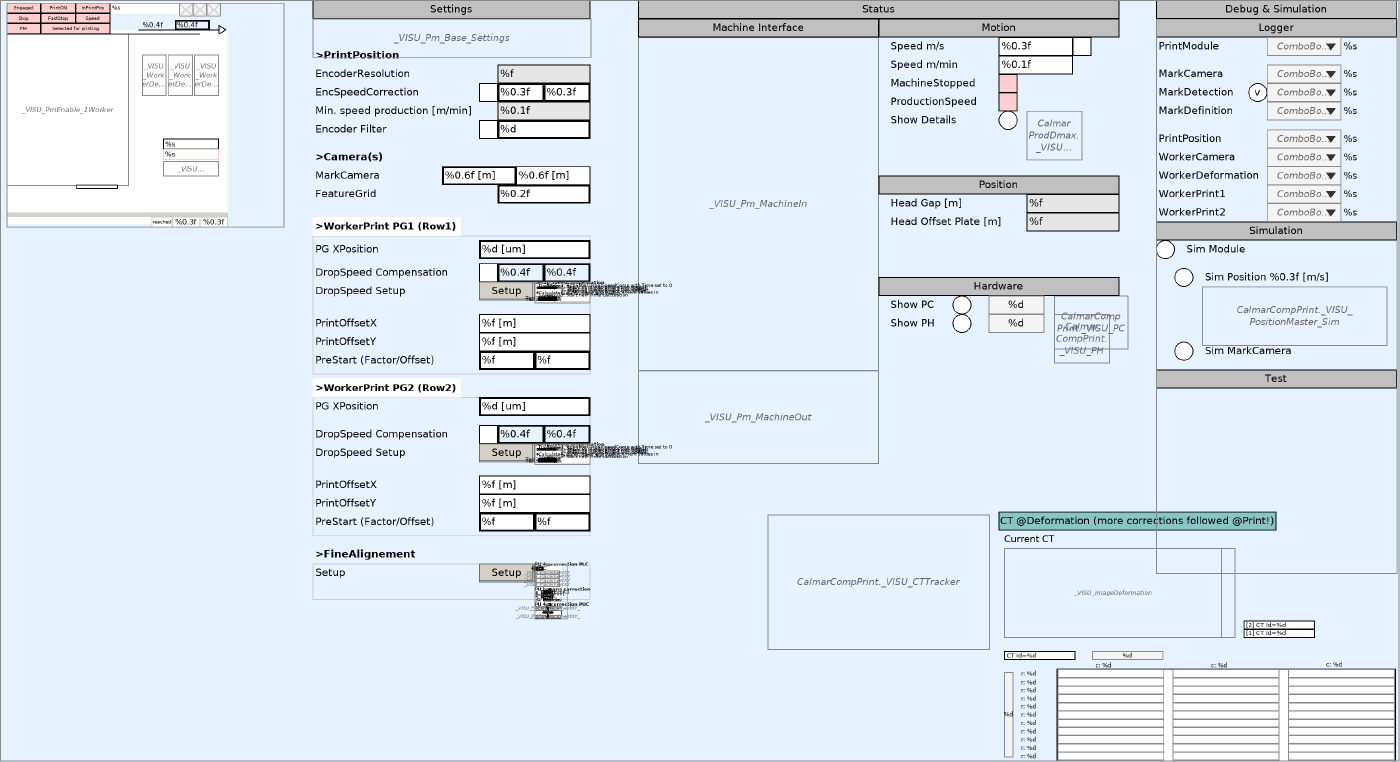
VISUALIZATION _VISU_Pm_WEU_1Worker  // 1514x825
VAR_IN_OUT
  mInst : FB_PrintModule_WEU;
END_VAR
    Frame (1086,574 428x251)
        shows _VISU_CT_Details(mInst := mInst.fbWorkerPrint[1])
    Rectangle (1080,554 300x20), "CT @Deformation (more corrections followed @Print!)"
    Frame (1140,320 80x58), invisible if: NOT mInst.fbView.bShowPcDetail
        shows CalmarCompPrint._VISU_PC(mInst := mInst._pPc[mInst.fbView.nSelPcDetail]^)
    Rectangle (960,340 110x20), "Show PH"
    Rectangle (960,320 110x20), "Show PC"
    Rectangle (960,40 120x20), "Speed m/s"
    Rectangle (1080,40 80x20), "%0.3f", text variable: mInst.fSpeed
    RoundedRectangle (1080,80 20x20), colour toggle: mInst.bMoving
    Rectangle (960,80 110x20), "MachineStopped"
    RoundedRectangle (1080,100 20x20), colour toggle: mInst.bSpeedReachedForPrinting
    Rectangle (960,100 110x20), "ProductionSpeed"
    Rectangle (960,60 120x20), "Speed m/min"
    Rectangle (1080,60 80x20), "%0.1f", text variable: mInst.fSpeedMpMin
    RoundedRectangle (1160,40 20x20), tooltip "Exeeds max. speed=%f", colour toggle: mInst._pModuleMachineFeedback^.bSpeedExeeded
        p4168582468: mInst._pModuleMachineFeedback^.fMaxSpeed
    Frame (690,401 260x101)
        shows _VISU_Pm_MachineOut(ref := mInst._pModuleMachineFeedback^)
    Frame (690,40 260x361)
        shows _VISU_Pm_MachineIn(ref := mInst._pModuleMachineState^)
    Rectangle (690,20 260x20), "Machine Interface"
    Rectangle (950,20 260x20), "Motion"
    Frame (7,3 300x243)
        shows _VISU_Pm_WEU_mini_1Worker(mInst := mInst)
    Rectangle (960,120 110x20), "Show Details"
    Ellipse (1080,120 20x20)
        toggle mInst.fbView.bShowPositionDetail
    Ellipse (1030,340 20x20)
        toggle mInst.fbView.bShowPhDetail
    Rectangle (950,300 260x20), "Hardware"
    Ellipse (1030,320 20x20)
        toggle mInst.fbView.bShowPcDetail
    Frame (1250,20 261x601), invisible if: NOT mInst.fbView.bShowDebugAndSim
        shows _VISU_Pm_WEU_Debug(mInst := mInst)
    Rectangle (338,0 300x20), "Settings"
    Rectangle (690,0 520x20), "Status"
    Rectangle (1250,0 260x20), "Debug & Simulation"
        toggle mInst.fbView.bShowDebugAndSim
    Rectangle (950,190 260x20), "Position"
    Rectangle (960,230 140x20), "Head Offset Plate [m]"
    Rectangle (1110,230 100x20), "%f", text variable: mInst.fC_HeadOffsetPlate
    Frame (1110,120 60x53), invisible if: NOT mInst.fbView.bShowPositionDetail
        shows CalmarProdDmax._VISU_PrintPositionDmax(m_Inst := mInst.fbPrintPosition)
    Frame (1140,340 60x53), invisible if: NOT mInst.fbView.bShowPhDetail
        shows CalmarCompPrint._VISU_PH(mInst := mInst._pPh[mInst.fbView.nSelPhDetail]^)
    Scrollbar (1069,340 60x20), "%d", text variable: mInst.fbView.nSelPhDetail, invisible if: NOT mInst.fbView.bShowPhDetail
        p2245068023: mInst._nPh
        p1057716461: mInst.fbView.nSelPhDetail
    Scrollbar (1069,320 60x20), "%d", text variable: mInst.fbView.nSelPcDetail, invisible if: NOT mInst.fbView.bShowPcDetail
        p2245068023: mInst._nPc
        p1057716461: mInst.fbView.nSelPcDetail
    Rectangle (1110,210 100x20), "%f", text variable: mInst._pModuleMachineFeedback^.fHeadGap
    Rectangle (960,210 140x20), "Head Gap [m]"
    Frame (338,20 299x522)
        shows _VISU_Pm_WEU_Settings(mInst := mInst)
    Frame (830,557 240x146)
        shows CalmarCompPrint._VISU_CTTracker(mInst := mInst.fbCTTracker)
END_VISUALIZATION

// ---- POUs/Print/WEU/_VISU_Pm_WEU_mini.TcVIS
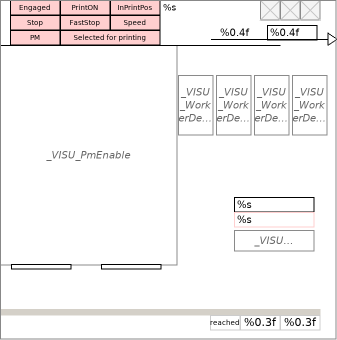
VISUALIZATION _VISU_Pm_WEU_mini  // 337x340
VAR_IN_OUT
  mInst : FB_PrintModule_WEU;
END_VAR
    Rectangle (160,0 160x15), "%s", text variable: mInst.fbAdsPm.stAds.aO_Name
    Rectangle (0,60 330x280)
    RoundedRectangle (0,309 320x6), colour toggle: mInst.fbView.bMovingInd
    Frame (0,45 177x220)
        shows _VISU_PmEnable(mInst := mInst)
        p2738717112: mInst.fbView.zPos_PM
    RoundedRectangle (11,264 60x5), colour toggle: mInst.fbView.bPrintInd[2]
        p2738717112: mInst.fbView.zPos_PM
    RoundedRectangle (101,264 60x5), colour toggle: mInst.fbView.bPrintInd[1]
        p2738717112: mInst.fbView.zPos_PM
    Line (0,45) (280,45)
    Frame (254,75 35x60)
        shows _VISU_WorkerDefGrid_small(m_Inst := mInst.fbWorkerDeformation)
    Frame (292,75 35x60)
        shows _VISU_WorkerDefGrid_small(m_Inst := mInst.fbWorkerCamera)
    Frame (178,75 35x60)
        shows _VISU_WorkerDefGrid_small(m_Inst := mInst.fbWorkerPrint[2])
    Frame (216,75 35x60)
        shows _VISU_WorkerDefGrid_small(m_Inst := mInst.fbWorkerPrint[1])
    Frame (234,230 80x21)
        shows _VISU_MarkDetection_Trigger(mInst := mInst.fbMarkCameraWeu.fbMarkDetection)
    Rectangle (234,197 80x15), "%s", tooltip "active camera device", text variable: mInst.fbWorkerCamera._iActiveCam.sName
    Rectangle (234,212 80x15), "%s", tooltip "active camera mode", text variable: mInst.fbWorkerCamera._iActiveCam.eCameraMode, colour toggle: mInst.fbWorkerCamera._bCamValid
    Rectangle (217,25 50x15), "%0.4f", tooltip "PM position on main tracker", text variable: mInst._fPmMainTrackPos
    Polyline (211,39) (328,39) (328,33) (337,39) (328,45) (328,39)
    RoundedRectangle (10,30 50x15), "PM"
        toggle mInst.fbAdsPm.stAds.bI_Enable
    RoundedRectangle (10,0 50x15), "Engaged", colour toggle: mInst._pModuleMachineState^.bEngaged
    RoundedRectangle (60,0 50x15), "PrintON", colour toggle: mInst._pModuleMachineState^.bPrintActivated
    RoundedRectangle (110,0 50x15), "InPrintPos", colour toggle: mInst._pModuleMachineState^.bUnitInPrintPosition
    RoundedRectangle (10,15 50x15), "Stop", colour toggle: NOT mInst._pModuleMachineState^.bStopRequest
    RoundedRectangle (60,15 50x15), "FastStop", colour toggle: NOT mInst._pModuleMachineState^.bFastStopRequest
    RoundedRectangle (110,15 50x15), "Speed", colour toggle: mInst.bSpeedReachedForPrinting
    RoundedRectangle (280,315 40x15), "%0.3f", tooltip "Target speed", text variable: mInst._pModuleMachineState^.fTargetSpeed
    RoundedRectangle (240,315 40x15), "%0.3f", tooltip "Current Speed", text variable: mInst.fSpeed
    RoundedRectangle (210,315 30x15), "reached", tooltip "Target speed reached", colour toggle: mInst._pModuleMachineState^.bTargetSpeedReached
    Image (260,0 20x20), invisible if: NOT mInst._pModuleMachineState^.bSleep, image: ImagePool_Steinemann.sleep_icon
    Image (280,0 20x20), invisible if: NOT mInst._pModuleMachineState^.bShutdown, image: ImagePool_Steinemann.shutdown_icon
    Image (300,0 20x20), invisible if: NOT mInst._pModuleMachineState^.bEStop, image: ImagePool_Steinemann.estop_icon
    Rectangle (267,25 50x15), "%0.4f", tooltip "PM position to previous", text variable: mInst._fPmDistToPrev
    RoundedRectangle (60,30 100x15), "Selected for printing"
        toggle mInst.bSelectedForPrint
END_VISUALIZATION

// ---- POUs/Print/WEU/_VISU_Pm_WEU_mini_1Worker.TcVIS
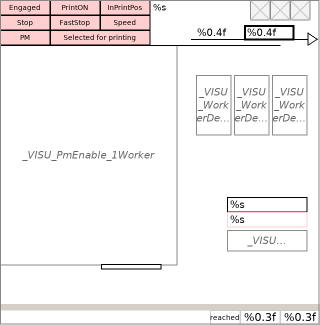
VISUALIZATION _VISU_Pm_WEU_mini_1Worker  // 320x325
VAR_IN_OUT
  mInst : FB_PrintModule_WEU;
END_VAR
    Rectangle (150,0 160x15), "%s", text variable: mInst.fbAdsPm.stAds.aO_Name
    Rectangle (0,40 320x280)
    Frame (227,230 80x21)
        shows _VISU_MarkDetection_Trigger(mInst := mInst.fbMarkDetection)
    Rectangle (227,197 80x15), "%s", tooltip "active camera device", text variable: mInst.fbWorkerCamera._iActiveCam.sName
    Rectangle (227,212 80x15), "%s", tooltip "active camera mode", text variable: mInst.fbWorkerCamera._iActiveCam.eCameraMode, colour toggle: mInst.fbWorkerCamera._bCamValid
    RoundedRectangle (0,304 320x6), colour toggle: mInst.fbView.bMovingInd
    Frame (0,45 177x220)
        shows _VISU_PmEnable_1Worker(mInst := mInst)
        p2738717112: mInst.fbView.zPos_PM
    RoundedRectangle (101,264 60x5), colour toggle: mInst.fbView.bPrintInd[1]
        p2738717112: mInst.fbView.zPos_PM
    Line (0,45) (280,45)
    RoundedRectangle (280,310 40x15), "%0.3f", tooltip "Target speed", text variable: mInst._pModuleMachineState^.fTargetSpeed
    RoundedRectangle (240,310 40x15), "%0.3f", tooltip "Current Speed", text variable: mInst.fSpeed
    RoundedRectangle (0,0 50x15), "Engaged", colour toggle: mInst._pModuleMachineState^.bEngaged
    RoundedRectangle (50,0 50x15), "PrintON", colour toggle: mInst._pModuleMachineState^.bPrintActivated
    RoundedRectangle (100,0 50x15), "InPrintPos", colour toggle: mInst._pModuleMachineState^.bUnitInPrintPosition
    RoundedRectangle (0,15 50x15), "Stop", colour toggle: NOT mInst._pModuleMachineState^.bStopRequest
    RoundedRectangle (50,15 50x15), "FastStop", colour toggle: NOT mInst._pModuleMachineState^.bFastStopRequest
    RoundedRectangle (100,15 50x15), "Speed", colour toggle: mInst.bSpeedReachedForPrinting
    Image (250,0 20x20), invisible if: NOT mInst._pModuleMachineState^.bSleep, image: ImagePool_Steinemann.sleep_icon
    Image (270,0 20x20), invisible if: NOT mInst._pModuleMachineState^.bShutdown, image: ImagePool_Steinemann.shutdown_icon
    Image (290,0 20x20), invisible if: NOT mInst._pModuleMachineState^.bEStop, image: ImagePool_Steinemann.estop_icon
    RoundedRectangle (210,310 30x15), "reached", tooltip "Target speed reached", colour toggle: mInst._pModuleMachineState^.bTargetSpeedReached
    Frame (234,75 35x60)
        shows _VISU_WorkerDefGrid_small(m_Inst := mInst.fbWorkerDeformation)
    Frame (272,75 35x60)
        shows _VISU_WorkerDefGrid_small(m_Inst := mInst.fbWorkerCamera)
    Frame (196,75 35x60)
        shows _VISU_WorkerDefGrid_small(m_Inst := mInst.fbWorkerPrint[1])
    RoundedRectangle (50,30 100x15), "Selected for printing"
        toggle mInst.bSelectedForPrint
    RoundedRectangle (0,30 50x15), "PM"
        toggle mInst.fbAdsPm.stAds.bI_Enable
    Rectangle (194,25 50x15), "%0.4f", tooltip "PM position on main tracker", text variable: mInst._fPmMainTrackPos
    Polyline (191,39) (308,39) (308,33) (317,39) (308,45) (308,39)
    Rectangle (244,25 50x15), "%0.4f", tooltip "PM position to previous", text variable: mInst._fPmDistToPrev
        OnMouseClick: write the text variable via Default
END_VISUALIZATION

// ---- POUs/Print/WEU/_VISU_Pm_WEU_Worker.TcVIS
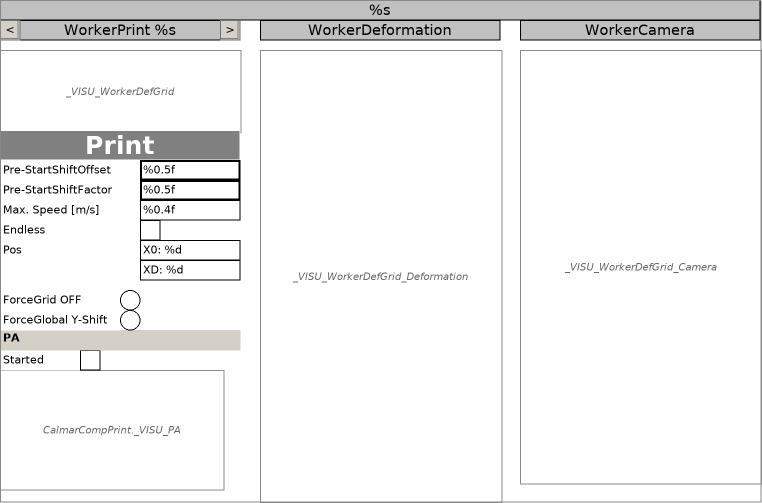
VISUALIZATION _VISU_Pm_WEU_Worker  // 762x503
VAR_IN_OUT
	mInst : FB_PrintModule_WEU;
END_VAR
    Frame (0,50 242x406)
        shows _VISU_WorkerPrint_WEU(m_Inst := mInst.fbWorkerPrint[mInst.fbView.nSelWorkerPrint])
    Rectangle (0,20 240x20), "WorkerPrint %s", text variable: mInst.fbView.nSelWorkerPrint
    Frame (520,50 242x434)
        shows _VISU_WorkerDefGrid_Camera(m_Inst := mInst.fbWorkerCamera)
    Rectangle (520,20 240x20), "WorkerCamera"
    Rectangle (0,0 760x20), "%s", text variable: mInst.fbAdsPm.aO_Name
    Rectangle (260,20 240x20), "WorkerDeformation"
    Frame (260,50 242x453)
        shows _VISU_WorkerDefGrid_Deformation(m_Inst := mInst.fbWorkerDeformation)
    Button (0,20 20x20), "<"
        OnMouseClick: execute { mInst.fbView.nSelWorkerPrint := mInst.fbView.nSelWorkerPrint - 1; }
    Button (220,20 20x20), ">"
        OnMouseClick: execute { mInst.fbView.nSelWorkerPrint := mInst.fbView.nSelWorkerPrint + 1; }
END_VISUALIZATION

// ---- POUs/Print/WEU/_VISU_WorkerPrint_WEU.TcVIS
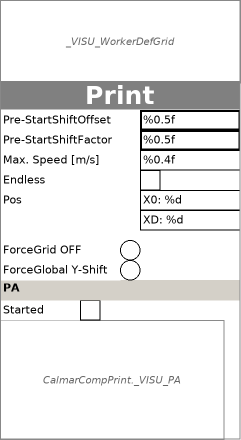
VISUALIZATION _VISU_WorkerPrint_WEU  // 241x440
VAR_IN_OUT
  m_Inst : FB_WorkerDefGrid_Print_WEU;
END_VAR
    Frame (0,0 241x83)
        shows _VISU_WorkerDefGrid(m_Inst := m_Inst)
    Rectangle (0,80 240x30), "Print", colour toggle: m_Inst._pAttachedCt <> 0
    Frame (0,320 224x120)
        shows CalmarCompPrint._VISU_PA(m_Inst := m_Inst.fbPa)
    Rectangle (0,150 120x20), "Max. Speed [m/s]"
    Rectangle (140,150 100x20), "%0.4f", text variable: m_Inst.fMaxSpeed
    Rectangle (0,170 120x20), "Endless"
    RoundedRectangle (140,170 20x20), colour toggle: m_Inst._bEndless
    Rectangle (0,300 80x20), "Started"
    RoundedRectangle (80,300 20x20), colour toggle: m_Inst._bPaStarted
    Rectangle (0,190 120x20), "Pos"
    Rectangle (140,190 100x20), "X0: %d", text variable: m_Inst._nPosX0
    Rectangle (140,210 100x20), "XD: %d", text variable: m_Inst._nPosXDelta
    Rectangle (0,280 240x20), "PA"
    Rectangle (0,240 120x20), "ForceGrid OFF"
    Ellipse (120,240 20x20), tooltip "Force Grid OFF (gridPs=0)"
        toggle m_Inst._bForceDefGridOff
    Rectangle (0,110 160x20), "Pre-StartShiftOffset"
    Rectangle (140,110 100x20), "%0.5f", text variable: m_Inst._fStartShiftOffset
        OnMouseDown: write the text variable via Default
    Rectangle (0,130 160x20), "Pre-StartShiftFactor"
    Rectangle (140,130 100x20), "%0.5f", text variable: m_Inst._fStartShiftFactor
        OnMouseDown: write the text variable via Default
    Rectangle (0,260 120x20), "ForceGlobal Y-Shift"
    Ellipse (120,260 20x20), tooltip "Force Grid OFF (gridPs=0)"
        toggle m_Inst._bForceGlobalYShift
END_VISUALIZATION
